C07324=1151.022,358.801,-80.777,-176.348,9.228,148.809
C07325=1151.025,358.554,-80.742,-176.350,9.224,148.808
C07326=1151.029,358.306,-80.708,-176.353,9.220,148.808
C07327=1151.034,358.059,-80.672,-176.355,9.216,148.807
C07328=1151.038,357.811,-80.638,-176.358,9.212,148.807
C07329=1151.041,357.564,-80.602,-176.361,9.208,148.807
C07330=1151.045,357.317,-80.568,-176.363,9.205,148.807
C07331=1151.049,357.068,-80.533,-176.365,9.201,148.806
C07332=1151.053,356.822,-80.498,-176.368,9.196,148.806
C07333=1151.057,356.573,-80.463,-176.370,9.193,148.806
C07334=1151.062,356.326,-80.429,-176.373,9.189,148.805
C07335=1151.065,356.079,-80.394,-176.375,9.185,148.805
C07336=1151.069,355.831,-80.359,-176.378,9.181,148.805
C07337=1151.073,355.583,-80.325,-176.380,9.178,148.804
C07338=1151.076,355.336,-80.290,-176.383,9.173,148.804
C07339=1151.081,355.089,-80.255,-176.386,9.169,148.804
C07340=1151.085,354.841,-80.220,-176.388,9.166,148.804
C07341=1151.089,354.593,-80.186,-176.390,9.162,148.803
C07342=1151.093,354.345,-80.152,-176.393,9.158,148.803
C07343=1151.097,354.099,-80.116,-176.396,9.154,148.803
C07344=1151.101,353.850,-80.082,-176.398,9.151,148.802
C07345=1151.105,353.603,-80.048,-176.400,9.147,148.802
C07346=1151.109,353.355,-80.013,-176.403,9.143,148.802
C07347=1151.113,353.108,-79.978,-176.405,9.139,148.801
C07348=1151.116,352.860,-79.944,-176.408,9.135,148.801
C07349=1151.121,352.613,-79.910,-176.410,9.132,148.801
C07350=1151.124,352.365,-79.875,-176.413,9.127,148.800
C07351=1151.128,352.118,-79.840,-176.415,9.124,148.800
C07352=1151.132,351.870,-79.805,-176.418,9.120,148.800
C07353=1151.136,351.623,-79.772,-176.420,9.116,148.799
C07354=1151.140,351.375,-79.737,-176.423,9.112,148.799
C07355=1151.144,351.127,-79.703,-176.425,9.109,148.799
C07356=1151.149,350.880,-79.668,-176.428,9.105,148.799
C07357=1151.153,350.632,-79.634,-176.431,9.100,148.798
C07358=1151.156,350.385,-79.600,-176.433,9.097,148.798
C07359=1151.160,350.137,-79.565,-176.436,9.093,148.798
C07360=1151.164,349.890,-79.531,-176.438,9.089,148.797
C07361=1151.168,349.641,-79.496,-176.441,9.085,148.797
C07362=1151.172,349.394,-79.463,-176.443,9.082,148.797
C07363=1151.177,349.146,-79.429,-176.446,9.078,148.797
C07364=1151.180,348.899,-79.394,-176.448,9.074,148.796
C07365=1151.185,348.651,-79.360,-176.451,9.070,148.796
C07366=1151.188,348.403,-79.326,-176.453,9.067,148.796
C07367=1151.193,348.156,-79.291,-176.456,9.063,148.796
C07368=1151.196,347.909,-79.257,-176.458,9.059,148.795
C07369=1151.201,347.660,-79.223,-176.461,9.055,148.795
C07370=1151.204,347.413,-79.189,-176.463,9.052,148.795
C07371=1151.209,347.166,-79.155,-176.466,9.048,148.794
C07372=1151.212,346.918,-79.121,-176.468,9.044,148.794
C07373=1151.216,346.670,-79.087,-176.471,9.040,148.794
C07374=1151.221,346.423,-79.053,-176.473,9.037,148.794
C07375=1151.224,346.175,-79.019,-176.476,9.033,148.793
C07376=1151.229,345.927,-78.984,-176.478,9.029,148.793
C07377=1151.233,345.680,-78.951,-176.481,9.025,148.793
C07378=1151.236,345.432,-78.917,-176.483,9.022,148.792
C07379=1151.241,345.184,-78.882,-176.486,9.018,148.792
C07380=1151.245,344.937,-78.849,-176.488,9.014,148.792
C07381=1151.248,344.689,-78.815,-176.491,9.010,148.792
C07382=1151.253,344.441,-78.781,-176.493,9.007,148.791
C07383=1151.257,344.194,-78.747,-176.496,9.003,148.791
C07384=1151.261,343.947,-78.714,-176.498,8.999,148.791
C07385=1151.265,343.698,-78.679,-176.501,8.995,148.790
C07386=1151.269,343.451,-78.646,-176.503,8.992,148.790
C07387=1151.273,343.203,-78.612,-176.506,8.988,148.790
C07388=1151.277,342.955,-78.578,-176.508,8.984,148.790
C07389=1151.281,342.707,-78.544,-176.511,8.980,148.789
C07390=1151.285,342.460,-78.511,-176.514,8.977,148.789
C07391=1151.289,342.212,-78.477,-176.516,8.973,148.789
C07392=1151.293,341.964,-78.443,-176.518,8.969,148.789
C07393=1151.297,341.716,-78.409,-176.521,8.965,148.788
C07394=1151.301,341.469,-78.376,-176.524,8.962,148.788
C07395=1151.305,341.222,-78.342,-176.527,8.958,148.788
C07396=1151.310,340.974,-78.308,-176.529,8.955,148.788
C07397=1151.313,340.726,-78.274,-176.531,8.950,148.787
C07398=1151.317,340.478,-78.241,-176.534,8.947,148.787
C07399=1151.321,340.231,-78.207,-176.536,8.944,148.787
C07400=1151.325,339.983,-78.174,-176.539,8.940,148.787
C07401=1151.330,339.703,-78.136,-176.542,8.936,148.786
C07402=1151.335,339.423,-78.098,-176.545,8.931,148.786
C07403=1151.339,339.142,-78.060,-176.548,8.927,148.786
C07404=1151.344,338.863,-78.022,-176.550,8.923,148.785
C07405=1151.347,338.614,-77.989,-176.553,8.919,148.785
C07406=1151.352,338.367,-77.955,-176.555,8.916,148.785
C07407=1151.355,338.120,-77.922,-176.558,8.912,148.785
C07408=1151.360,337.871,-77.888,-176.560,8.908,148.785
C07409=1151.364,337.624,-77.855,-176.563,8.905,148.784
C07410=1151.369,337.376,-77.822,-176.566,8.901,148.784
C07411=1151.372,337.128,-77.787,-176.568,8.898,148.784
C07412=1151.376,336.880,-77.754,-176.571,8.893,148.784
C07413=1151.380,336.633,-77.721,-176.573,8.890,148.783
C07414=1151.384,336.385,-77.688,-176.575,8.887,148.783
C07415=1151.388,336.137,-77.655,-176.578,8.883,148.783
C07416=1151.392,335.890,-77.622,-176.580,8.879,148.783
C07417=1151.397,335.642,-77.588,-176.583,8.875,148.782
C07418=1151.401,335.394,-77.555,-176.586,8.872,148.782
C07419=1151.405,335.147,-77.521,-176.588,8.868,148.782
C07420=1151.408,334.899,-77.488,-176.591,8.865,148.782
C07421=1151.412,334.651,-77.455,-176.593,8.861,148.782
C07422=1151.416,334.403,-77.422,-176.596,8.857,148.781
C07423=1151.421,334.155,-77.388,-176.598,8.854,148.781
C07424=1151.425,333.908,-77.355,-176.601,8.850,148.781
C07425=1151.429,333.660,-77.322,-176.604,8.847,148.781
C07426=1151.433,333.412,-77.289,-176.606,8.842,148.780
C07427=1151.437,333.164,-77.256,-176.609,8.839,148.780
C07428=1151.440,332.917,-77.223,-176.611,8.836,148.780
C07429=1151.445,332.669,-77.190,-176.614,8.831,148.780
C07430=1151.449,332.421,-77.158,-176.616,8.828,148.779
C07431=1151.453,332.173,-77.124,-176.619,8.824,148.779
C07432=1151.457,331.926,-77.091,-176.621,8.821,148.779
C07433=1151.461,331.678,-77.058,-176.623,8.818,148.779
C07434=1151.466,331.430,-77.025,-176.626,8.813,148.778
C07435=1151.470,331.182,-76.992,-176.629,8.810,148.778
C07436=1151.473,330.935,-76.959,-176.632,8.806,148.778
C07437=1151.478,330.687,-76.927,-176.634,8.803,148.778
C07438=1151.482,330.439,-76.894,-176.636,8.800,148.778
C07439=1151.486,330.191,-76.860,-176.639,8.795,148.777
C07440=1151.490,329.943,-76.827,-176.641,8.792,148.777
C07441=1151.494,329.696,-76.794,-176.644,8.788,148.777
C07442=1151.498,329.448,-76.762,-176.647,8.785,148.777
C07443=1151.502,329.200,-76.729,-176.649,8.782,148.777
C07444=1151.506,328.952,-76.696,-176.652,8.777,148.776
C07445=1151.511,328.704,-76.664,-176.654,8.774,148.776
C07446=1151.514,328.456,-76.631,-176.657,8.770,148.776
C07447=1151.518,328.209,-76.598,-176.659,8.767,148.776
C07448=1151.523,327.960,-76.565,-176.662,8.764,148.775
C07449=1151.527,327.713,-76.532,-176.665,8.759,148.775
C07450=1151.530,327.465,-76.500,-176.667,8.757,148.775
C07451=1151.535,327.217,-76.467,-176.670,8.753,148.775
C07452=1151.539,326.969,-76.434,-176.673,8.749,148.775
C07453=1151.543,326.722,-76.402,-176.675,8.746,148.775
C07454=1151.547,326.474,-76.369,-176.678,8.742,148.774
C07455=1151.551,326.226,-76.336,-176.680,8.739,148.774
C07456=1151.556,325.978,-76.304,-176.682,8.735,148.774
C07457=1151.559,325.731,-76.271,-176.685,8.731,148.774
C07458=1151.564,325.482,-76.239,-176.688,8.728,148.774
C07459=1151.567,325.235,-76.206,-176.690,8.725,148.773
C07460=1151.571,324.986,-76.174,-176.693,8.721,148.773
C07461=1151.576,324.739,-76.141,-176.695,8.717,148.773
C07462=1151.580,324.491,-76.109,-176.698,8.714,148.773
C07463=1151.584,324.244,-76.076,-176.700,8.710,148.773
C07464=1151.588,323.996,-76.044,-176.703,8.707,148.772
C07465=1151.592,323.747,-76.012,-176.706,8.704,148.772
C07466=1151.596,323.499,-75.979,-176.708,8.700,148.772
C07467=1151.600,323.251,-75.947,-176.711,8.696,148.772
C07468=1151.604,323.004,-75.914,-176.713,8.693,148.772
C07469=1151.608,322.756,-75.882,-176.716,8.689,148.771
C07470=1151.613,322.508,-75.850,-176.718,8.686,148.771
C07471=1151.616,322.261,-75.817,-176.721,8.682,148.771
C07472=1151.621,322.012,-75.785,-176.723,8.678,148.771
C07473=1151.624,321.764,-75.753,-176.726,8.675,148.771
C07474=1151.629,321.516,-75.720,-176.729,8.671,148.771
C07475=1151.633,321.269,-75.688,-176.731,8.668,148.770
C07476=1151.637,321.021,-75.656,-176.734,8.665,148.770
C07477=1151.641,320.773,-75.624,-176.737,8.661,148.770
C07478=1151.645,320.525,-75.591,-176.739,8.657,148.770
C07479=1151.649,320.278,-75.559,-176.741,8.654,148.770
C07480=1151.654,320.029,-75.527,-176.744,8.651,148.769
C07481=1151.658,319.781,-75.495,-176.747,8.647,148.769
C07482=1151.661,319.533,-75.463,-176.749,8.644,148.769
C07483=1151.665,319.286,-75.430,-176.752,8.640,148.769
C07484=1151.670,319.038,-75.399,-176.755,8.636,148.769
C07485=1151.674,318.790,-75.366,-176.757,8.633,148.769
C07486=1151.678,318.542,-75.334,-176.759,8.630,148.768
C07487=1151.682,318.294,-75.302,-176.762,8.626,148.768
C07488=1151.687,318.046,-75.270,-176.765,8.623,148.768
C07489=1151.690,317.798,-75.238,-176.767,8.619,148.768
C07490=1151.694,317.550,-75.207,-176.770,8.615,148.768
C07491=1151.699,317.302,-75.175,-176.772,8.612,148.768
C07492=1151.703,317.054,-75.143,-176.775,8.609,148.767
C07493=1151.707,316.806,-75.111,-176.778,8.605,148.767
C07494=1151.712,316.559,-75.079,-176.780,8.602,148.767
C07495=1151.715,316.311,-75.047,-176.783,8.599,148.767
C07496=1151.719,316.063,-75.015,-176.785,8.595,148.767
C07497=1151.723,315.814,-74.983,-176.788,8.591,148.767
C07498=1151.728,315.567,-74.951,-176.791,8.588,148.767
C07499=1151.731,315.319,-74.919,-176.793,8.585,148.766
C07500=1151.736,315.071,-74.887,-176.796,8.581,148.766
C07501=1151.740,314.823,-74.855,-176.798,8.578,148.766
C07502=1151.744,314.575,-74.824,-176.801,8.575,148.766
C07503=1151.748,314.328,-74.792,-176.804,8.571,148.766
C07504=1151.753,314.079,-74.760,-176.806,8.567,148.766
C07505=1151.757,313.802,-74.724,-176.809,8.563,148.765
C07506=1151.762,313.524,-74.689,-176.812,8.560,148.765
C07507=1151.767,313.247,-74.654,-176.815,8.556,148.765
C07508=1151.771,312.969,-74.618,-176.818,8.552,148.765
C07509=1151.775,312.721,-74.586,-176.820,8.549,148.765
C07510=1151.780,312.474,-74.554,-176.823,8.545,148.765
C07511=1151.784,312.225,-74.523,-176.826,8.542,148.765
C07512=1151.788,311.978,-74.492,-176.828,8.538,148.764
C07513=1151.792,311.730,-74.460,-176.830,8.535,148.764
C07514=1151.796,311.481,-74.429,-176.834,8.531,148.764
C07515=1151.800,311.234,-74.397,-176.836,8.528,148.764
C07516=1151.804,310.986,-74.365,-176.838,8.525,148.764
C07517=1151.809,310.738,-74.333,-176.841,8.522,148.764
C07518=1151.813,310.489,-74.302,-176.844,8.518,148.764
C07519=1151.817,310.242,-74.271,-176.846,8.515,148.763
C07520=1151.821,309.993,-74.240,-176.849,8.511,148.763
C07521=1151.825,309.745,-74.208,-176.852,8.507,148.763
C07522=1151.829,309.498,-74.176,-176.854,8.504,148.763
C07523=1151.833,309.249,-74.145,-176.856,8.501,148.763
C07524=1151.837,309.002,-74.114,-176.859,8.498,148.763
C07525=1151.841,308.753,-74.083,-176.862,8.494,148.763
C07526=1151.846,308.506,-74.051,-176.864,8.491,148.762
C07527=1151.850,308.257,-74.020,-176.867,8.488,148.763
C07528=1151.854,308.010,-73.989,-176.870,8.484,148.762
C07529=1151.858,307.761,-73.957,-176.872,8.480,148.762
C07530=1151.862,307.514,-73.926,-176.875,8.477,148.762
C07531=1151.866,307.265,-73.895,-176.878,8.474,148.762
C07532=1151.871,307.018,-73.863,-176.880,8.471,148.762
C07533=1151.875,306.769,-73.832,-176.883,8.467,148.762
C07534=1151.879,306.522,-73.801,-176.886,8.464,148.762
C07535=1151.884,306.274,-73.770,-176.888,8.460,148.761
C07536=1151.887,306.026,-73.738,-176.891,8.458,148.761
C07537=1151.892,305.778,-73.707,-176.893,8.454,148.761
C07538=1151.896,305.529,-73.676,-176.896,8.450,148.761
C07539=1151.900,305.282,-73.645,-176.899,8.447,148.761
C07540=1151.904,305.033,-73.614,-176.901,8.444,148.761
C07541=1151.909,304.785,-73.583,-176.903,8.441,148.761
C07542=1151.913,304.537,-73.551,-176.907,8.437,148.761
C07543=1151.917,304.289,-73.520,-176.909,8.434,148.760
C07544=1151.922,304.041,-73.489,-176.911,8.430,148.760
C07545=1151.925,303.794,-73.458,-176.914,8.427,148.760
C07546=1151.929,303.546,-73.427,-176.917,8.423,148.760
C07547=1151.933,303.297,-73.396,-176.920,8.420,148.760
C07548=1151.938,303.049,-73.366,-176.922,8.417,148.760
C07549=1151.942,302.802,-73.334,-176.924,8.414,148.760
C07550=1151.946,302.553,-73.303,-176.927,8.411,148.760
C07551=1151.951,302.305,-73.272,-176.930,8.407,148.760
C07552=1151.955,302.058,-73.242,-176.933,8.404,148.760
C07553=1151.959,301.809,-73.211,-176.935,8.401,148.759
C07554=1151.963,301.561,-73.180,-176.937,8.397,148.759
C07555=1151.968,301.314,-73.149,-176.940,8.394,148.759
C07556=1151.972,301.065,-73.118,-176.943,8.390,148.759
C07557=1151.976,300.817,-73.087,-176.946,8.387,148.759
C07558=1151.980,300.569,-73.056,-176.948,8.384,148.759
C07559=1151.984,300.321,-73.025,-176.950,8.381,148.759
C07560=1151.989,300.073,-72.995,-176.953,8.378,148.759
C07561=1151.993,299.825,-72.965,-176.956,8.374,148.759
C07562=1151.997,299.576,-72.933,-176.959,8.371,148.759
C07563=1152.001,299.328,-72.903,-176.961,8.367,148.758
C07564=1152.005,299.081,-72.872,-176.964,8.365,148.758
C07565=1152.009,298.832,-72.841,-176.966,8.361,148.758
C07566=1152.014,298.584,-72.811,-176.970,8.357,148.758
C07567=1152.018,298.337,-72.780,-176.972,8.354,148.758
C07568=1152.022,298.088,-72.749,-176.974,8.351,148.758
C07569=1152.026,297.840,-72.718,-176.977,8.348,148.758
C07570=1152.030,297.592,-72.688,-176.979,8.345,148.758
C07571=1152.035,297.344,-72.658,-176.983,8.341,148.758
C07572=1152.039,297.096,-72.626,-176.985,8.338,148.758
C07573=1152.043,296.848,-72.596,-176.988,8.335,148.758
C07574=1152.047,296.600,-72.565,-176.990,8.331,148.757
C07575=1152.052,296.351,-72.535,-176.993,8.328,148.757
C07576=1152.056,296.103,-72.505,-176.995,8.325,148.757
C07577=1152.060,295.855,-72.474,-176.998,8.321,148.757
C07578=1152.064,295.608,-72.444,-177.001,8.318,148.757
C07579=1152.069,295.360,-72.413,-177.004,8.315,148.757
C07580=1152.072,295.111,-72.383,-177.006,8.312,148.757
C07581=1152.077,294.863,-72.353,-177.009,8.309,148.757
C07582=1152.081,294.615,-72.322,-177.012,8.305,148.757
C07583=1152.085,294.367,-72.292,-177.014,8.302,148.757
C07584=1152.089,294.118,-72.261,-177.017,8.299,148.757
C07585=1152.094,293.870,-72.231,-177.019,8.296,148.757
C07586=1152.098,293.622,-72.200,-177.022,8.292,148.757
C07587=1152.102,293.375,-72.170,-177.024,8.290,148.757
C07588=1152.106,293.126,-72.141,-177.027,8.286,148.756
C07589=1152.111,292.878,-72.110,-177.030,8.282,148.756
C07590=1152.114,292.630,-72.079,-177.032,8.279,148.756
C07591=1152.119,292.381,-72.049,-177.035,8.276,148.756
C07592=1152.123,292.134,-72.019,-177.038,8.273,148.756
C07593=1152.127,291.886,-71.988,-177.040,8.270,148.756
C07594=1152.132,291.637,-71.959,-177.043,8.267,148.756
C07595=1152.136,291.390,-71.928,-177.046,8.263,148.756
C07596=1152.140,291.141,-71.898,-177.049,8.260,148.756
C07597=1152.144,290.893,-71.868,-177.051,8.257,148.756
C07598=1152.149,290.644,-71.838,-177.054,8.254,148.756
C07599=1152.153,290.397,-71.808,-177.056,8.251,148.756
C07600=1152.157,290.148,-71.778,-177.059,8.248,148.756
C07601=1152.161,289.900,-71.748,-177.061,8.244,148.756
C07602=1152.165,289.652,-71.718,-177.065,8.241,148.756
C07603=1152.170,289.404,-71.688,-177.067,8.238,148.756
C07604=1152.174,289.156,-71.658,-177.070,8.234,148.755
C07605=1152.178,288.908,-71.628,-177.072,8.231,148.755
C07606=1152.182,288.659,-71.598,-177.075,8.228,148.755
C07607=1152.186,288.411,-71.567,-177.077,8.225,148.755
C07608=1152.191,288.163,-71.538,-177.080,8.222,148.755
C07609=1152.195,287.888,-71.505,-177.083,8.218,148.755
C07610=1152.201,287.613,-71.471,-177.086,8.215,148.755
C07611=1152.205,287.337,-71.438,-177.089,8.211,148.755
C07612=1152.210,287.062,-71.405,-177.092,8.207,148.755
C07613=1152.214,286.814,-71.375,-177.095,8.204,148.755
C07614=1152.218,286.566,-71.346,-177.097,8.201,148.755
C07615=1152.223,286.317,-71.315,-177.100,8.198,148.755
C07616=1152.227,286.070,-71.285,-177.103,8.195,148.755
C07617=1152.231,285.821,-71.256,-177.105,8.192,148.755
C07618=1152.235,285.573,-71.226,-177.108,8.189,148.755
C07619=1152.239,285.325,-71.197,-177.110,8.186,148.755
C07620=1152.244,285.077,-71.166,-177.114,8.182,148.755
C07621=1152.248,284.829,-71.137,-177.116,8.179,148.755
C07622=1152.252,284.580,-71.107,-177.119,8.176,148.755
C07623=1152.256,284.332,-71.078,-177.121,8.173,148.755
C07624=1152.261,284.084,-71.048,-177.124,8.170,148.755
C07625=1152.266,283.835,-71.018,-177.126,8.167,148.754
C07626=1152.269,283.588,-70.988,-177.129,8.164,148.754
C07627=1152.274,283.339,-70.959,-177.132,8.161,148.755
C07628=1152.278,283.091,-70.929,-177.134,8.157,148.754
C07629=1152.282,282.843,-70.900,-177.137,8.154,148.754
C07630=1152.286,282.595,-70.870,-177.140,8.151,148.754
C07631=1152.290,282.346,-70.841,-177.143,8.147,148.754
C07632=1152.294,282.098,-70.811,-177.146,8.145,148.754
C07633=1152.300,281.850,-70.782,-177.148,8.142,148.754
C07634=1152.304,281.602,-70.752,-177.151,8.138,148.754
C07635=1152.308,281.354,-70.723,-177.153,8.135,148.754
C07636=1152.313,281.105,-70.693,-177.156,8.132,148.754
C07637=1152.317,280.857,-70.664,-177.158,8.129,148.754
C07638=1152.321,280.609,-70.634,-177.161,8.126,148.754
C07639=1152.325,280.361,-70.605,-177.164,8.123,148.754
C07640=1152.329,280.112,-70.576,-177.166,8.120,148.754
C07641=1152.333,279.864,-70.546,-177.170,8.116,148.754
C07642=1152.338,279.616,-70.517,-177.172,8.113,148.754
C07643=1152.342,279.367,-70.487,-177.175,8.110,148.754
C07644=1152.347,279.120,-70.458,-177.178,8.107,148.754
C07645=1152.351,278.872,-70.429,-177.180,8.104,148.754
C07646=1152.355,278.623,-70.399,-177.183,8.101,148.754
C07647=1152.359,278.375,-70.370,-177.185,8.098,148.754
C07648=1152.364,278.126,-70.341,-177.188,8.095,148.754
C07649=1152.368,277.878,-70.312,-177.191,8.092,148.754
C07650=1152.372,277.630,-70.282,-177.193,8.089,148.754
C07651=1152.377,277.382,-70.253,-177.196,8.086,148.754
C07652=1152.380,277.134,-70.224,-177.199,8.083,148.754
C07653=1152.385,276.885,-70.195,-177.202,8.080,148.754
C07654=1152.389,276.637,-70.166,-177.204,8.077,148.754
C07655=1152.393,276.389,-70.137,-177.207,8.074,148.754
C07656=1152.397,276.140,-70.107,-177.210,8.070,148.754
C07657=1152.402,275.892,-70.079,-177.213,8.067,148.754
C07658=1152.407,275.644,-70.049,-177.215,8.064,148.754
C07659=1152.411,275.396,-70.020,-177.218,8.061,148.754
C07660=1152.414,275.148,-69.991,-177.221,8.058,148.754
C07661=1152.419,274.899,-69.962,-177.223,8.055,148.754
C07662=1152.423,274.651,-69.933,-177.226,8.052,148.754
C07663=1152.428,274.402,-69.904,-177.229,8.049,148.754
C07664=1152.432,274.154,-69.875,-177.231,8.046,148.754
C07665=1152.436,273.906,-69.845,-177.234,8.043,148.754
C07666=1152.441,273.658,-69.818,-177.236,8.039,148.754
C07667=1152.445,273.410,-69.788,-177.239,8.037,148.754
C07668=1152.449,273.161,-69.759,-177.242,8.034,148.754
C07669=1152.453,272.913,-69.730,-177.245,8.031,148.754
C07670=1152.457,272.665,-69.702,-177.247,8.027,148.754
C07671=1152.462,272.416,-69.673,-177.250,8.024,148.754
C07672=1152.466,272.168,-69.643,-177.253,8.022,148.754
C07673=1152.471,271.919,-69.615,-177.255,8.019,148.754
C07674=1152.475,271.672,-69.586,-177.258,8.016,148.754
C07675=1152.479,271.423,-69.557,-177.260,8.012,148.754
C07676=1152.483,271.175,-69.528,-177.263,8.009,148.754
C07677=1152.488,270.927,-69.500,-177.266,8.006,148.754
C07678=1152.492,270.678,-69.471,-177.269,8.004,148.754
C07679=1152.496,270.430,-69.442,-177.272,8.001,148.754
C07680=1152.501,270.182,-69.414,-177.274,7.997,148.754
C07681=1152.505,269.934,-69.385,-177.277,7.994,148.754
C07682=1152.509,269.685,-69.356,-177.279,7.991,148.754
C07683=1152.514,269.437,-69.328,-177.282,7.988,148.754
C07684=1152.518,269.189,-69.299,-177.285,7.986,148.754
C07685=1152.522,268.940,-69.270,-177.288,7.983,148.754
C07686=1152.527,268.692,-69.242,-177.290,7.979,148.754
C07687=1152.531,268.444,-69.213,-177.293,7.976,148.754
C07688=1152.535,268.195,-69.184,-177.296,7.973,148.754
C07689=1152.540,267.947,-69.156,-177.299,7.970,148.754
C07690=1152.544,267.699,-69.127,-177.302,7.967,148.754
C07691=1152.548,267.450,-69.099,-177.304,7.964,148.754
C07692=1152.553,267.202,-69.070,-177.307,7.961,148.754
C07693=1152.557,266.953,-69.042,-177.310,7.958,148.754
C07694=1152.561,266.706,-69.013,-177.312,7.955,148.754
C07695=1152.566,266.457,-68.984,-177.315,7.952,148.754
C07696=1152.570,266.208,-68.956,-177.318,7.949,148.754
C07697=1152.575,265.960,-68.928,-177.320,7.947,148.754
C07698=1152.578,265.711,-68.900,-177.323,7.944,148.754
C07699=1152.584,265.463,-68.871,-177.325,7.940,148.754
C07700=1152.587,265.215,-68.842,-177.328,7.938,148.754
C07701=1152.592,264.967,-68.814,-177.331,7.935,148.754
C07702=1152.596,264.719,-68.786,-177.333,7.932,148.754
C07703=1152.600,264.470,-68.757,-177.336,7.929,148.754
C07704=1152.605,264.222,-68.729,-177.339,7.926,148.755
C07705=1152.609,263.973,-68.701,-177.342,7.923,148.755
C07706=1152.613,263.725,-68.673,-177.345,7.920,148.755
C07707=1152.618,263.476,-68.644,-177.347,7.917,148.755
C07708=1152.622,263.228,-68.616,-177.350,7.914,148.755
C07709=1152.626,262.980,-68.588,-177.352,7.911,148.755
C07710=1152.631,262.732,-68.560,-177.355,7.908,148.755
C07711=1152.635,262.483,-68.532,-177.358,7.905,148.755
C07712=1152.640,262.235,-68.503,-177.361,7.902,148.755
C07713=1152.645,261.961,-68.473,-177.364,7.898,148.755
C07714=1152.649,261.689,-68.441,-177.367,7.895,148.755
C07715=1152.654,261.415,-68.411,-177.370,7.892,148.755
C07716=1152.659,261.142,-68.379,-177.373,7.888,148.755
C07717=1152.663,260.893,-68.351,-177.376,7.886,148.755
C07718=1152.667,260.645,-68.323,-177.379,7.883,148.755
C07719=1152.672,260.396,-68.295,-177.381,7.880,148.755
C07720=1152.676,260.148,-68.268,-177.384,7.877,148.755
C07721=1152.680,259.899,-68.239,-177.386,7.875,148.755
C07722=1152.685,259.651,-68.211,-177.389,7.872,148.755
C07723=1152.689,259.403,-68.183,-177.392,7.869,148.755
C07724=1152.693,259.155,-68.155,-177.394,7.865,148.755
C07725=1152.698,258.906,-68.126,-177.397,7.863,148.755
C07726=1152.702,258.657,-68.099,-177.400,7.860,148.755
C07727=1152.707,258.409,-68.072,-177.403,7.857,148.755
C07728=1152.711,258.161,-68.043,-177.405,7.854,148.756
C07729=1152.716,257.913,-68.015,-177.408,7.851,148.756
C07730=1152.720,257.663,-67.988,-177.411,7.848,148.756
C07731=1152.724,257.416,-67.960,-177.414,7.845,148.756
C07732=1152.728,257.167,-67.932,-177.416,7.842,148.756
C07733=1152.732,256.919,-67.905,-177.419,7.839,148.756
C07734=1152.737,256.670,-67.876,-177.422,7.836,148.756
C07735=1152.741,256.422,-67.848,-177.425,7.833,148.756
C07736=1152.746,256.173,-67.821,-177.427,7.830,148.756
C07737=1152.750,255.925,-67.793,-177.430,7.827,148.756
C07738=1152.754,255.677,-67.765,-177.432,7.825,148.756
C07739=1152.759,255.428,-67.738,-177.435,7.822,148.756
C07740=1152.763,255.179,-67.709,-177.438,7.819,148.756
C07741=1152.768,254.931,-67.682,-177.441,7.816,148.756
C07742=1152.772,254.683,-67.655,-177.444,7.813,148.756
C07743=1152.776,254.434,-67.626,-177.446,7.810,148.757
C07744=1152.781,254.186,-67.599,-177.449,7.808,148.757
C07745=1152.785,253.938,-67.572,-177.452,7.805,148.757
C07746=1152.789,253.689,-67.544,-177.455,7.802,148.757
C07747=1152.793,253.441,-67.516,-177.457,7.799,148.757
C07748=1152.798,253.193,-67.489,-177.460,7.796,148.757
C07749=1152.802,252.944,-67.461,-177.463,7.793,148.757
C07750=1152.807,252.695,-67.434,-177.465,7.791,148.757
C07751=1152.811,252.447,-67.406,-177.468,7.788,148.757
C07752=1152.816,252.199,-67.379,-177.471,7.785,148.757
C07753=1152.820,251.950,-67.351,-177.474,7.782,148.757
C07754=1152.825,251.702,-67.323,-177.476,7.779,148.757
C07755=1152.829,251.453,-67.296,-177.479,7.776,148.757
C07756=1152.833,251.205,-67.268,-177.482,7.773,148.757
C07757=1152.838,250.956,-67.241,-177.485,7.770,148.757
C07758=1152.842,250.708,-67.214,-177.487,7.767,148.758
C07759=1152.847,250.460,-67.186,-177.490,7.764,148.758
C07760=1152.851,250.211,-67.159,-177.493,7.761,148.758
C07761=1152.855,249.962,-67.132,-177.495,7.759,148.758
C07762=1152.860,249.714,-67.104,-177.498,7.756,148.758
C07763=1152.864,249.466,-67.077,-177.501,7.753,148.758
C07764=1152.868,249.217,-67.050,-177.504,7.750,148.758
C07765=1152.872,248.968,-67.023,-177.506,7.748,148.758
C07766=1152.877,248.720,-66.995,-177.509,7.745,148.758
C07767=1152.881,248.472,-66.968,-177.512,7.742,148.758
C07768=1152.886,248.223,-66.941,-177.515,7.739,148.758
C07769=1152.890,247.974,-66.914,-177.517,7.737,148.759
C07770=1152.895,247.726,-66.887,-177.520,7.734,148.759
C07771=1152.899,247.478,-66.859,-177.523,7.731,148.759
C07772=1152.904,247.229,-66.832,-177.526,7.728,148.759
C07773=1152.908,246.981,-66.805,-177.528,7.725,148.759
C07774=1152.912,246.732,-66.778,-177.531,7.722,148.759
C07775=1152.916,246.484,-66.751,-177.534,7.719,148.759
C07776=1152.921,246.235,-66.724,-177.537,7.716,148.759
C07777=1152.926,245.987,-66.697,-177.539,7.714,148.759
C07778=1152.930,245.739,-66.669,-177.542,7.711,148.759
C07779=1152.935,245.490,-66.642,-177.544,7.708,148.759
C07780=1152.939,245.242,-66.616,-177.547,7.705,148.759
C07781=1152.943,244.993,-66.588,-177.550,7.703,148.759
C07782=1152.947,244.744,-66.561,-177.553,7.700,148.760
C07783=1152.952,244.496,-66.534,-177.556,7.697,148.760
C07784=1152.956,244.248,-66.508,-177.558,7.695,148.760
C07785=1152.960,243.999,-66.480,-177.561,7.692,148.760
C07786=1152.965,243.751,-66.453,-177.564,7.689,148.760
C07787=1152.970,243.502,-66.426,-177.567,7.686,148.760
C07788=1152.974,243.254,-66.400,-177.569,7.683,148.760
C07789=1152.978,243.005,-66.372,-177.572,7.680,148.760
C07790=1152.982,242.756,-66.345,-177.575,7.677,148.760
C07791=1152.987,242.508,-66.318,-177.578,7.675,148.761
C07792=1152.991,242.259,-66.293,-177.580,7.673,148.761
C07793=1152.996,242.010,-66.266,-177.583,7.670,148.761
C07794=1153.001,241.762,-66.238,-177.586,7.667,148.761
C07795=1153.005,241.514,-66.212,-177.589,7.664,148.761
C07796=1153.009,241.265,-66.185,-177.592,7.661,148.761
C07797=1153.014,241.017,-66.158,-177.594,7.659,148.761
C07798=1153.018,240.769,-66.131,-177.597,7.656,148.761
C07799=1153.023,240.519,-66.105,-177.600,7.653,148.762
C07800=1153.027,240.271,-66.078,-177.603,7.650,148.762
C07801=1153.031,240.023,-66.052,-177.605,7.647,148.762
C07802=1153.036,239.774,-66.024,-177.608,7.644,148.762
C07803=1153.040,239.526,-65.998,-177.610,7.642,148.762
C07804=1153.045,239.277,-65.972,-177.613,7.639,148.762
C07805=1153.050,239.029,-65.945,-177.616,7.636,148.762
C07806=1153.053,238.780,-65.918,-177.619,7.634,148.762
C07807=1153.058,238.531,-65.892,-177.622,7.631,148.762
C07808=1153.062,238.283,-65.865,-177.624,7.629,148.763
C07809=1153.067,238.035,-65.838,-177.627,7.626,148.763
C07810=1153.071,237.786,-65.812,-177.630,7.623,148.763
C07811=1153.076,237.537,-65.785,-177.632,7.620,148.763
C07812=1153.080,237.289,-65.759,-177.636,7.617,148.763
C07813=1153.085,237.040,-65.733,-177.638,7.615,148.763
C07814=1153.089,236.792,-65.706,-177.641,7.612,148.763
C07815=1153.093,236.543,-65.679,-177.643,7.609,148.763
C07816=1153.098,236.294,-65.653,-177.646,7.606,148.763
C07817=1153.103,236.023,-65.624,-177.649,7.604,148.764
C07818=1153.108,235.751,-65.595,-177.652,7.601,148.764
C07819=1153.112,235.479,-65.567,-177.655,7.598,148.764
C07820=1153.117,235.207,-65.537,-177.658,7.595,148.764
C07821=1153.121,234.958,-65.511,-177.661,7.592,148.764
C07822=1153.126,234.710,-65.484,-177.664,7.590,148.764
C07823=1153.131,234.462,-65.459,-177.667,7.587,148.764
C07824=1153.135,234.213,-65.432,-177.669,7.584,148.764
C07825=1153.140,233.964,-65.406,-177.672,7.582,148.765
C07826=1153.144,233.716,-65.379,-177.675,7.579,148.765
C07827=1153.148,233.467,-65.353,-177.678,7.576,148.765
C07828=1153.153,233.218,-65.327,-177.680,7.573,148.765
C07829=1153.157,232.970,-65.301,-177.683,7.571,148.765
C07830=1153.162,232.721,-65.274,-177.685,7.568,148.765
C07831=1153.166,232.473,-65.248,-177.689,7.565,148.766
C07832=1153.170,232.225,-65.223,-177.691,7.563,148.766
C07833=1153.175,231.976,-65.196,-177.694,7.560,148.766
C07834=1153.179,231.727,-65.170,-177.696,7.558,148.766
C07835=1153.183,231.479,-65.144,-177.700,7.555,148.766
C07836=1153.188,231.229,-65.118,-177.702,7.552,148.766
C07837=1153.192,230.981,-65.091,-177.705,7.549,148.766
C07838=1153.197,230.733,-65.066,-177.707,7.547,148.766
C07839=1153.202,230.484,-65.040,-177.710,7.544,148.766
C07840=1153.206,230.236,-65.013,-177.713,7.541,148.767
C07841=1153.210,229.987,-64.987,-177.716,7.539,148.767
C07842=1153.215,229.738,-64.961,-177.718,7.536,148.767
C07843=1153.219,229.489,-64.935,-177.721,7.533,148.767
C07844=1153.224,229.242,-64.909,-177.724,7.531,148.767
C07845=1153.228,228.993,-64.883,-177.727,7.528,148.767
C07846=1153.233,228.744,-64.857,-177.729,7.526,148.768
C07847=1153.237,228.495,-64.831,-177.732,7.523,148.768
C07848=1153.242,228.247,-64.806,-177.735,7.520,148.768
C07849=1153.246,227.998,-64.780,-177.738,7.517,148.768
C07850=1153.250,227.750,-64.754,-177.740,7.515,148.768
C07851=1153.255,227.501,-64.727,-177.743,7.512,148.768
C07852=1153.260,227.252,-64.702,-177.747,7.510,148.769
C07853=1153.264,227.004,-64.676,-177.749,7.508,148.769
C07854=1153.269,226.755,-64.650,-177.752,7.505,148.769
C07855=1153.273,226.506,-64.625,-177.754,7.502,148.769
C07856=1153.277,226.257,-64.599,-177.758,7.499,148.769
C07857=1153.282,226.009,-64.574,-177.760,7.497,148.769
C07858=1153.287,225.760,-64.547,-177.763,7.494,148.769
C07859=1153.291,225.511,-64.521,-177.766,7.492,148.770
C07860=1153.296,225.263,-64.496,-177.769,7.489,148.770
C07861=1153.300,225.014,-64.470,-177.771,7.487,148.770
C07862=1153.304,224.766,-64.445,-177.774,7.484,148.770
C07863=1153.309,224.517,-64.419,-177.777,7.481,148.770
C07864=1153.313,224.269,-64.393,-177.779,7.479,148.770
C07865=1153.318,224.020,-64.368,-177.782,7.476,148.770
C07866=1153.322,223.771,-64.342,-177.785,7.473,148.771
C07867=1153.327,223.523,-64.317,-177.787,7.471,148.771
C07868=1153.331,223.274,-64.291,-177.790,7.468,148.771
C07869=1153.335,223.025,-64.265,-177.793,7.466,148.771
C07870=1153.341,222.777,-64.239,-177.796,7.463,148.771
C07871=1153.345,222.528,-64.213,-177.798,7.461,148.771
C07872=1153.349,222.279,-64.188,-177.801,7.458,148.772
C07873=1153.354,222.031,-64.163,-177.804,7.455,148.772
C07874=1153.358,221.782,-64.137,-177.807,7.453,148.772
C07875=1153.363,221.533,-64.111,-177.809,7.450,148.772
C07876=1153.368,221.285,-64.086,-177.813,7.448,148.772
C07877=1153.371,221.036,-64.062,-177.815,7.445,148.772
C07878=1153.376,220.788,-64.036,-177.818,7.443,148.773
C07879=1153.380,220.539,-64.010,-177.821,7.440,148.773
C07880=1153.385,220.290,-63.985,-177.823,7.438,148.773
C07881=1153.389,220.042,-63.959,-177.826,7.435,148.773
C07882=1153.394,219.793,-63.934,-177.829,7.432,148.773
C07883=1153.399,219.545,-63.909,-177.831,7.430,148.774
C07884=1153.403,219.296,-63.883,-177.834,7.427,148.774
C07885=1153.408,219.046,-63.858,-177.837,7.425,148.774
C07886=1153.412,218.798,-63.833,-177.840,7.423,148.774
C07887=1153.417,218.549,-63.807,-177.842,7.420,148.774
C07888=1153.422,218.301,-63.782,-177.846,7.417,148.774
C07889=1153.425,218.052,-63.757,-177.848,7.415,148.775
C07890=1153.429,217.803,-63.731,-177.851,7.412,148.775
C07891=1153.435,217.555,-63.707,-177.854,7.410,148.775
C07892=1153.439,217.306,-63.681,-177.856,7.407,148.775
C07893=1153.444,217.057,-63.656,-177.859,7.404,148.775
C07894=1153.448,216.808,-63.631,-177.862,7.402,148.775
C07895=1153.452,216.561,-63.606,-177.864,7.400,148.776
C07896=1153.457,216.311,-63.581,-177.868,7.397,148.776
C07897=1153.462,216.063,-63.555,-177.870,7.394,148.776
C07898=1153.466,215.814,-63.530,-177.873,7.392,148.776
C07899=1153.471,215.565,-63.505,-177.876,7.390,148.776
C07900=1153.475,215.316,-63.480,-177.878,7.387,148.777
C07901=1153.480,215.068,-63.455,-177.881,7.385,148.777
C07902=1153.484,214.819,-63.430,-177.884,7.382,148.777
C07903=1153.489,214.571,-63.405,-177.886,7.380,148.777
C07904=1153.493,214.322,-63.380,-177.889,7.377,148.777
C07905=1153.498,214.073,-63.355,-177.892,7.374,148.778
C07906=1153.502,213.824,-63.330,-177.894,7.372,148.778
C07907=1153.506,213.576,-63.306,-177.898,7.370,148.778
C07908=1153.511,213.327,-63.280,-177.900,7.368,148.778
C07909=1153.516,213.078,-63.255,-177.903,7.365,148.778
C07910=1153.520,212.829,-63.230,-177.906,7.362,148.778
C07911=1153.524,212.581,-63.205,-177.908,7.360,148.779
C07912=1153.529,212.331,-63.180,-177.911,7.357,148.779
C07913=1153.534,212.083,-63.155,-177.914,7.354,148.779
C07914=1153.538,211.835,-63.131,-177.917,7.353,148.779
C07915=1153.543,211.586,-63.106,-177.920,7.350,148.779
C07916=1153.548,211.337,-63.081,-177.922,7.348,148.780
C07917=1153.551,211.088,-63.056,-177.925,7.345,148.780
C07918=1153.556,210.840,-63.031,-177.928,7.342,148.780
C07919=1153.560,210.590,-63.007,-177.931,7.340,148.780
C07920=1153.565,210.342,-62.982,-177.933,7.337,148.780
C07921=1153.570,210.072,-62.955,-177.937,7.335,148.781
C07922=1153.575,209.801,-62.928,-177.939,7.332,148.781
C07923=1153.580,209.531,-62.901,-177.942,7.330,148.781
C07924=1153.585,209.260,-62.875,-177.945,7.327,148.781
C07925=1153.590,209.012,-62.849,-177.948,7.325,148.782
C07926=1153.593,208.762,-62.825,-177.951,7.322,148.782
C07927=1153.599,208.514,-62.800,-177.954,7.320,148.782
C07928=1153.604,208.265,-62.776,-177.956,7.317,148.782
C07929=1153.607,208.016,-62.751,-177.959,7.315,148.782
C07930=1153.613,207.767,-62.726,-177.962,7.312,148.783
C07931=1153.617,207.519,-62.702,-177.964,7.310,148.783
C07932=1153.621,207.270,-62.677,-177.967,7.308,148.783
C07933=1153.626,207.022,-62.653,-177.970,7.305,148.783
C07934=1153.631,206.773,-62.628,-177.973,7.303,148.783
C07935=1153.635,206.524,-62.603,-177.976,7.300,148.784
C07936=1153.640,206.275,-62.579,-177.978,7.298,148.784
C07937=1153.644,206.027,-62.555,-177.981,7.295,148.784
C07938=1153.649,205.777,-62.530,-177.984,7.294,148.784
C07939=1153.653,205.529,-62.506,-177.987,7.291,148.784
C07940=1153.657,205.280,-62.482,-177.989,7.289,148.785
C07941=1153.663,205.032,-62.457,-177.992,7.286,148.785
C07942=1153.666,204.782,-62.432,-177.995,7.283,148.785
C07943=1153.671,204.534,-62.408,-177.998,7.281,148.785
C07944=1153.676,204.285,-62.384,-178.000,7.279,148.785
C07945=1153.680,204.036,-62.359,-178.003,7.277,148.786
C07946=1153.685,203.787,-62.335,-178.006,7.274,148.786
C07947=1153.689,203.538,-62.311,-178.008,7.272,148.786
C07948=1153.695,203.290,-62.287,-178.011,7.269,148.786
C07949=1153.698,203.041,-62.262,-178.014,7.267,148.787
C07950=1153.703,202.792,-62.238,-178.017,7.264,148.787
C07951=1153.708,202.543,-62.213,-178.019,7.263,148.787
C07952=1153.712,202.295,-62.189,-178.022,7.260,148.787
C07953=1153.716,202.046,-62.165,-178.025,7.257,148.788
C07954=1153.722,201.797,-62.141,-178.028,7.255,148.788
C07955=1153.726,201.548,-62.117,-178.031,7.253,148.788
C07956=1153.730,201.300,-62.093,-178.033,7.250,148.788
C07957=1153.735,201.051,-62.068,-178.036,7.248,148.789
C07958=1153.739,200.802,-62.044,-178.039,7.246,148.789
C07959=1153.744,200.553,-62.020,-178.042,7.243,148.789
C07960=1153.748,200.305,-61.996,-178.044,7.241,148.789
C07961=1153.753,200.056,-61.972,-178.047,7.239,148.789
C07962=1153.758,199.807,-61.947,-178.050,7.236,148.790
C07963=1153.762,199.558,-61.924,-178.053,7.234,148.790
C07964=1153.766,199.309,-61.900,-178.055,7.232,148.790
C07965=1153.771,199.061,-61.875,-178.058,7.229,148.790
C07966=1153.776,198.811,-61.852,-178.061,7.227,148.791
C07967=1153.781,198.563,-61.828,-178.064,7.224,148.791
C07968=1153.785,198.315,-61.803,-178.066,7.223,148.791
C07969=1153.789,198.065,-61.780,-178.069,7.220,148.791
C07970=1153.794,197.816,-61.755,-178.072,7.218,148.792
C07971=1153.799,197.567,-61.732,-178.075,7.215,148.792
C07972=1153.803,197.319,-61.708,-178.077,7.213,148.792
C07973=1153.808,197.070,-61.684,-178.080,7.210,148.792
C07974=1153.812,196.821,-61.660,-178.083,7.209,148.793
C07975=1153.818,196.573,-61.636,-178.086,7.206,148.793
C07976=1153.822,196.323,-61.612,-178.088,7.204,148.793
C07977=1153.826,196.074,-61.588,-178.092,7.201,148.793
C07978=1153.831,195.825,-61.564,-178.094,7.199,148.793
C07979=1153.835,195.577,-61.540,-178.097,7.197,148.794
C07980=1153.840,195.328,-61.517,-178.099,7.195,148.794
C07981=1153.844,195.080,-61.493,-178.103,7.192,148.794
C07982=1153.849,194.831,-61.470,-178.105,7.190,148.794
C07983=1153.853,194.582,-61.445,-178.108,7.187,148.795
C07984=1153.859,194.333,-61.422,-178.110,7.185,148.795
C07985=1153.863,194.084,-61.397,-178.114,7.183,148.795
C07986=1153.868,193.835,-61.374,-178.116,7.181,148.796
C07987=1153.872,193.587,-61.350,-178.119,7.178,148.796
C07988=1153.877,193.338,-61.327,-178.122,7.176,148.796
C07989=1153.882,193.089,-61.303,-178.124,7.174,148.796
C07990=1153.885,192.840,-61.279,-178.127,7.172,148.796
C07991=1153.890,192.591,-61.255,-178.130,7.170,148.797
C07992=1153.895,192.342,-61.232,-178.133,7.167,148.797
C07993=1153.899,192.093,-61.208,-178.135,7.165,148.797
C07994=1153.904,191.844,-61.185,-178.138,7.162,148.797
C07995=1153.909,191.595,-61.161,-178.141,7.161,148.798
C07996=1153.913,191.347,-61.137,-178.144,7.158,148.798
C07997=1153.918,191.098,-61.114,-178.146,7.156,148.798
C07998=1153.922,190.849,-61.091,-178.150,7.153,148.799
C07999=1153.927,190.600,-61.066,-178.152,7.151,148.799
C08000=1153.931,190.351,-61.043,-178.155,7.150,148.799
C08001=1153.936,190.102,-61.020,-178.157,7.147,148.799
C08002=1153.941,189.853,-60.996,-178.160,7.145,148.800
C08003=1153.946,189.604,-60.973,-178.163,7.142,148.800
C08004=1153.950,189.357,-60.950,-178.165,7.140,148.800
C08005=1153.955,189.108,-60.927,-178.169,7.138,148.800
C08006=1153.959,188.859,-60.903,-178.171,7.136,148.801
C08007=1153.964,188.610,-60.880,-178.174,7.134,148.801
C08008=1153.969,188.361,-60.856,-178.177,7.131,148.801
C08009=1153.973,188.112,-60.833,-178.179,7.129,148.801
C08010=1153.978,187.863,-60.809,-178.182,7.127,148.802
C08011=1153.982,187.614,-60.786,-178.185,7.125,148.802
C08012=1153.987,187.365,-60.762,-178.188,7.122,148.802
C08013=1153.991,187.116,-60.740,-178.191,7.120,148.802
C08014=1153.996,186.867,-60.716,-178.193,7.118,148.803
C08015=1154.001,186.618,-60.693,-178.196,7.115,148.803
C08016=1154.005,186.369,-60.669,-178.199,7.114,148.803
C08017=1154.010,186.120,-60.646,-178.202,7.111,148.804
C08018=1154.014,185.872,-60.624,-178.204,7.109,148.804
C08019=1154.019,185.623,-60.600,-178.207,7.107,148.804
C08020=1154.024,185.374,-60.577,-178.210,7.104,148.804
C08021=1154.029,185.125,-60.554,-178.212,7.103,148.805
C08022=1154.033,184.876,-60.530,-178.216,7.100,148.805
C08023=1154.037,184.627,-60.508,-178.218,7.098,148.805
C08024=1154.042,184.378,-60.484,-178.221,7.095,148.805
C08025=1154.047,184.109,-60.459,-178.224,7.094,148.806
C08026=1154.052,183.839,-60.433,-178.227,7.091,148.806
C08027=1154.057,183.570,-60.409,-178.230,7.089,148.806
C08028=1154.062,183.300,-60.384,-178.233,7.086,148.807
C08029=1154.067,183.051,-60.361,-178.236,7.084,148.807
C08030=1154.071,182.802,-60.338,-178.239,7.082,148.807
C08031=1154.076,182.553,-60.314,-178.241,7.080,148.807
C08032=1154.081,182.305,-60.292,-178.244,7.078,148.808
C08033=1154.085,182.056,-60.269,-178.247,7.076,148.808
C08034=1154.090,181.807,-60.246,-178.250,7.073,148.808
C08035=1154.094,181.558,-60.223,-178.252,7.071,148.809
C08036=1154.098,181.309,-60.200,-178.255,7.069,148.809
C08037=1154.104,181.061,-60.177,-178.258,7.066,148.809
C08038=1154.109,180.811,-60.154,-178.260,7.065,148.809
C08039=1154.113,180.562,-60.132,-178.263,7.063,148.810
C08040=1154.117,180.313,-60.108,-178.266,7.060,148.810
C08041=1154.121,180.065,-60.085,-178.269,7.058,148.810
C08042=1154.127,179.816,-60.063,-178.271,7.057,148.811
C08043=1154.132,179.567,-60.040,-178.275,7.054,148.811
C08044=1154.136,179.318,-60.017,-178.277,7.052,148.811
C08045=1154.141,179.068,-59.994,-178.280,7.049,148.811
C08046=1154.145,178.820,-59.972,-178.283,7.048,148.812
C08047=1154.150,178.571,-59.949,-178.285,7.045,148.812
C08048=1154.154,178.322,-59.926,-178.288,7.043,148.812
C08049=1154.159,178.073,-59.903,-178.291,7.041,148.813
C08050=1154.164,177.824,-59.880,-178.294,7.039,148.813
C08051=1154.168,177.575,-59.858,-178.296,7.037,148.813
C08052=1154.173,177.326,-59.835,-178.299,7.035,148.814
C08053=1154.177,177.077,-59.812,-178.302,7.033,148.814
C08054=1154.183,176.828,-59.790,-178.305,7.030,148.814
C08055=1154.187,176.580,-59.767,-178.307,7.028,148.814
C08056=1154.192,176.330,-59.744,-178.310,7.027,148.815
C08057=1154.196,176.082,-59.722,-178.313,7.024,148.815
C08058=1154.201,175.833,-59.699,-178.316,7.022,148.815
C08059=1154.205,175.584,-59.677,-178.318,7.020,148.816
C08060=1154.210,175.336,-59.654,-178.321,7.018,148.816
C08061=1154.215,175.086,-59.631,-178.324,7.016,148.816
C08062=1154.219,174.837,-59.609,-178.326,7.014,148.816
C08063=1154.224,174.588,-59.586,-178.330,7.011,148.817
C08064=1154.228,174.340,-59.564,-178.332,7.010,148.817
C08065=1154.233,174.090,-59.541,-178.335,7.008,148.818
C08066=1154.238,173.842,-59.519,-178.338,7.005,148.818
C08067=1154.243,173.592,-59.496,-178.341,7.003,148.818
C08068=1154.247,173.343,-59.474,-178.343,7.001,148.818
C08069=1154.252,173.095,-59.452,-178.347,6.999,148.819
C08070=1154.257,172.845,-59.429,-178.349,6.997,148.819
C08071=1154.261,172.596,-59.406,-178.351,6.995,148.819
C08072=1154.266,172.348,-59.384,-178.354,6.993,148.820
C08073=1154.271,172.098,-59.362,-178.357,6.991,148.820
C08074=1154.275,171.850,-59.339,-178.360,6.989,148.820
C08075=1154.279,171.601,-59.317,-178.362,6.987,148.821
C08076=1154.284,171.351,-59.295,-178.366,6.984,148.821
C08077=1154.289,171.103,-59.272,-178.368,6.983,148.821
C08078=1154.293,170.854,-59.250,-178.371,6.981,148.821
C08079=1154.299,170.605,-59.228,-178.374,6.978,148.822
C08080=1154.303,170.356,-59.205,-178.376,6.976,148.822
C08081=1154.307,170.107,-59.183,-178.379,6.974,148.822
C08082=1154.313,169.858,-59.161,-178.382,6.973,148.823
C08083=1154.317,169.609,-59.139,-178.385,6.970,148.823
C08084=1154.322,169.360,-59.116,-178.387,6.968,148.823
C08085=1154.327,169.111,-59.094,-178.390,6.966,148.824
C08086=1154.331,168.862,-59.072,-178.393,6.964,148.824
C08087=1154.336,168.613,-59.050,-178.396,6.962,148.824
C08088=1154.341,168.364,-59.028,-178.398,6.960,148.825
C08089=1154.345,168.115,-59.005,-178.401,6.958,148.825
C08090=1154.350,167.867,-58.983,-178.404,6.956,148.825
C08091=1154.354,167.617,-58.961,-178.407,6.954,148.826
C08092=1154.359,167.368,-58.939,-178.409,6.952,148.826
C08093=1154.364,167.119,-58.918,-178.412,6.950,148.826
C08094=1154.369,166.870,-58.895,-178.415,6.948,148.827
C08095=1154.373,166.621,-58.873,-178.418,6.946,148.827
C08096=1154.377,166.372,-58.851,-178.421,6.944,148.827
C08097=1154.382,166.124,-58.829,-178.423,6.941,148.827
C08098=1154.387,165.875,-58.807,-178.426,6.939,148.828
C08099=1154.391,165.626,-58.785,-178.429,6.938,148.828
C08100=1154.397,165.377,-58.763,-178.431,6.936,148.829
C08101=1154.401,165.127,-58.741,-178.435,6.933,148.829
C08102=1154.406,164.879,-58.719,-178.437,6.932,148.829
C08103=1154.410,164.629,-58.697,-178.440,6.930,148.829
C08104=1154.415,164.381,-58.675,-178.442,6.928,148.830
C08105=1154.419,164.131,-58.653,-178.446,6.925,148.830
C08106=1154.424,163.883,-58.632,-178.448,6.924,148.831
C08107=1154.429,163.633,-58.610,-178.451,6.922,148.831
C08108=1154.434,163.385,-58.588,-178.453,6.920,148.831
C08109=1154.438,163.135,-58.566,-178.456,6.918,148.831
C08110=1154.443,162.887,-58.544,-178.459,6.915,148.832
C08111=1154.448,162.638,-58.522,-178.462,6.914,148.832
C08112=1154.453,162.388,-58.500,-178.465,6.912,148.833
C08113=1154.457,162.140,-58.478,-178.467,6.910,148.833
C08114=1154.462,161.890,-58.457,-178.471,6.908,148.833
C08115=1154.467,161.641,-58.435,-178.473,6.906,148.833
C08116=1154.471,161.392,-58.413,-178.476,6.904,148.834
C08117=1154.476,161.143,-58.391,-178.478,6.902,148.834
C08118=1154.481,160.895,-58.370,-178.481,6.900,148.835
C08119=1154.485,160.645,-58.348,-178.484,6.898,148.835
C08120=1154.490,160.396,-58.327,-178.487,6.896,148.835
C08121=1154.495,160.147,-58.305,-178.489,6.894,148.835
C08122=1154.499,159.898,-58.283,-178.492,6.892,148.836
C08123=1154.504,159.649,-58.261,-178.495,6.890,148.836
C08124=1154.509,159.400,-58.239,-178.498,6.888,148.837
C08125=1154.513,159.151,-58.219,-178.500,6.886,148.837
C08126=1154.518,158.902,-58.197,-178.503,6.885,148.837
C08127=1154.522,158.653,-58.175,-178.506,6.883,148.838
C08128=1154.527,158.404,-58.153,-178.509,6.880,148.838
C08129=1154.532,158.135,-58.130,-178.512,6.879,148.838
C08130=1154.537,157.866,-58.107,-178.515,6.876,148.839
C08131=1154.542,157.597,-58.083,-178.518,6.874,148.839
C08132=1154.547,157.328,-58.061,-178.521,6.873,148.840
C08133=1154.552,157.079,-58.040,-178.524,6.870,148.840
C08134=1154.557,156.830,-58.018,-178.526,6.868,148.840
C08135=1154.561,156.581,-57.996,-178.529,6.866,148.840
C08136=1154.567,156.332,-57.975,-178.531,6.864,148.841
C08137=1154.572,156.083,-57.953,-178.534,6.863,148.841
C08138=1154.576,155.835,-57.932,-178.537,6.860,148.842
C08139=1154.580,155.585,-57.911,-178.540,6.858,148.842
C08140=1154.585,155.336,-57.889,-178.543,6.857,148.842
C08141=1154.590,155.087,-57.868,-178.546,6.855,148.843
C08142=1154.595,154.838,-57.846,-178.548,6.853,148.843
C08143=1154.600,154.588,-57.825,-178.551,6.851,148.843
C08144=1154.604,154.340,-57.804,-178.554,6.849,148.844
C08145=1154.609,154.091,-57.782,-178.556,6.847,148.844
C08146=1154.613,153.841,-57.761,-178.559,6.845,148.844
C08147=1154.618,153.593,-57.739,-178.562,6.843,148.845
C08148=1154.623,153.343,-57.718,-178.565,6.842,148.845
C08149=1154.627,153.095,-57.697,-178.567,6.840,148.845
C08150=1154.633,152.846,-57.676,-178.571,6.837,148.846
C08151=1154.637,152.596,-57.655,-178.573,6.836,148.846
C08152=1154.642,152.347,-57.633,-178.576,6.834,148.847
C08153=1154.647,152.098,-57.613,-178.578,6.832,148.847
C08154=1154.651,151.850,-57.591,-178.581,6.830,148.847
C08155=1154.656,151.600,-57.570,-178.584,6.828,148.847
C08156=1154.660,151.351,-57.549,-178.587,6.826,148.848
C08157=1154.665,151.102,-57.528,-178.590,6.824,148.848
C08158=1154.670,150.853,-57.507,-178.592,6.822,148.849
C08159=1154.675,150.604,-57.485,-178.595,6.821,148.849
C08160=1154.680,150.355,-57.465,-178.598,6.819,148.849
C08161=1154.684,150.105,-57.443,-178.600,6.817,148.850
C08162=1154.689,149.857,-57.422,-178.603,6.816,148.850
C08163=1154.694,149.608,-57.401,-178.606,6.813,148.851
C08164=1154.699,149.358,-57.380,-178.609,6.811,148.851
C08165=1154.703,149.110,-57.359,-178.612,6.810,148.851
C08166=1154.708,148.861,-57.338,-178.615,6.808,148.852
C08167=1154.713,148.611,-57.317,-178.617,6.806,148.852
C08168=1154.717,148.362,-57.297,-178.619,6.804,148.852
C08169=1154.722,148.113,-57.275,-178.622,6.802,148.853
C08170=1154.727,147.864,-57.254,-178.625,6.801,148.853
C08171=1154.732,147.615,-57.234,-178.628,6.798,148.853
C08172=1154.737,147.366,-57.213,-178.631,6.796,148.854
C08173=1154.741,147.118,-57.192,-178.634,6.795,148.854
C08174=1154.746,146.868,-57.171,-178.636,6.793,148.854
C08175=1154.750,146.619,-57.150,-178.639,6.791,148.855
C08176=1154.755,146.369,-57.129,-178.642,6.789,148.855
C08177=1154.760,146.120,-57.109,-178.644,6.788,148.856
C08178=1154.765,145.871,-57.088,-178.647,6.786,148.856
C08179=1154.770,145.623,-57.066,-178.650,6.784,148.856
C08180=1154.774,145.374,-57.046,-178.653,6.782,148.857
C08181=1154.779,145.124,-57.025,-178.656,6.780,148.857
C08182=1154.784,144.875,-57.004,-178.659,6.778,148.858
C08183=1154.789,144.626,-56.983,-178.661,6.776,148.858
C08184=1154.793,144.377,-56.963,-178.664,6.775,148.858
C08185=1154.798,144.128,-56.942,-178.667,6.773,148.859
C08186=1154.803,143.879,-56.922,-178.669,6.771,148.859
C08187=1154.807,143.630,-56.901,-178.672,6.770,148.859
C08188=1154.812,143.381,-56.880,-178.675,6.768,148.860
C08189=1154.816,143.131,-56.859,-178.677,6.766,148.860
C08190=1154.821,142.882,-56.838,-178.680,6.764,148.861
C08191=1154.826,142.633,-56.818,-178.683,6.762,148.861
C08192=1154.831,142.384,-56.797,-178.686,6.760,148.861
C08193=1154.836,142.135,-56.777,-178.689,6.758,148.862
C08194=1154.840,141.886,-56.756,-178.692,6.757,148.862
C08195=1154.845,141.636,-56.735,-178.694,6.755,148.863
C08196=1154.850,141.388,-56.715,-178.697,6.753,148.863
C08197=1154.855,141.138,-56.694,-178.700,6.752,148.863
C08198=1154.859,140.889,-56.674,-178.702,6.750,148.864
C08199=1154.864,140.640,-56.653,-178.705,6.748,148.864
C08200=1154.869,140.391,-56.632,-178.708,6.746,148.865
C08201=1154.873,140.142,-56.612,-178.711,6.745,148.865
C08202=1154.878,139.893,-56.592,-178.713,6.743,148.865
C08203=1154.883,139.644,-56.571,-178.716,6.741,148.866
C08204=1154.888,139.394,-56.551,-178.719,6.740,148.866
C08205=1154.892,139.145,-56.531,-178.721,6.738,148.866
C08206=1154.898,138.897,-56.510,-178.725,6.735,148.867
C08207=1154.902,138.648,-56.490,-178.727,6.734,148.867
C08208=1154.907,138.399,-56.469,-178.730,6.732,148.868
C08209=1154.912,138.149,-56.449,-178.733,6.730,148.868
C08210=1154.917,137.900,-56.429,-178.736,6.728,148.868
C08211=1154.921,137.651,-56.408,-178.738,6.727,148.869
C08212=1154.926,137.402,-56.387,-178.741,6.725,148.869
C08213=1154.931,137.153,-56.367,-178.744,6.723,148.870
C08214=1154.935,136.903,-56.347,-178.746,6.721,148.870
C08215=1154.940,136.654,-56.327,-178.749,6.720,148.870
C08216=1154.945,136.405,-56.306,-178.752,6.718,148.871
C08217=1154.950,136.156,-56.286,-178.754,6.716,148.871
C08218=1154.954,135.907,-56.266,-178.757,6.715,148.872
C08219=1154.959,135.658,-56.246,-178.760,6.713,148.872
C08220=1154.964,135.410,-56.226,-178.763,6.711,148.872
C08221=1154.969,135.160,-56.205,-178.765,6.709,148.873
C08222=1154.974,134.911,-56.185,-178.768,6.708,148.873
C08223=1154.978,134.661,-56.165,-178.771,6.706,148.873
C08224=1154.983,134.412,-56.145,-178.773,6.704,148.874
C08225=1154.987,134.163,-56.125,-178.776,6.703,148.874
C08226=1154.993,133.913,-56.104,-178.779,6.701,148.875
C08227=1154.998,133.665,-56.084,-178.782,6.699,148.875
C08228=1155.002,133.416,-56.064,-178.784,6.697,148.875
C08229=1155.007,133.167,-56.044,-178.787,6.696,148.876
C08230=1155.011,132.918,-56.024,-178.790,6.694,148.876
C08231=1155.016,132.668,-56.004,-178.792,6.692,148.877
C08232=1155.020,132.419,-55.984,-178.796,6.691,148.877
C08233=1155.026,132.150,-55.962,-178.799,6.688,148.878
C08234=1155.032,131.882,-55.941,-178.802,6.687,148.878
C08235=1155.037,131.614,-55.919,-178.804,6.685,148.878
C08236=1155.042,131.345,-55.898,-178.807,6.683,148.879
C08237=1155.046,131.096,-55.878,-178.810,6.682,148.879
C08238=1155.051,130.847,-55.858,-178.813,6.680,148.880
C08239=1155.056,130.598,-55.838,-178.816,6.678,148.880
C08240=1155.061,130.348,-55.817,-178.818,6.677,148.881
C08241=1155.066,130.099,-55.798,-178.821,6.675,148.881
C08242=1155.071,129.850,-55.778,-178.824,6.673,148.881
C08243=1155.076,129.600,-55.758,-178.827,6.672,148.882
C08244=1155.080,129.352,-55.738,-178.829,6.670,148.882
C08245=1155.085,129.103,-55.718,-178.832,6.668,148.883
C08246=1155.090,128.853,-55.699,-178.835,6.666,148.883
C08247=1155.094,128.604,-55.678,-178.837,6.665,148.883
C08248=1155.099,128.355,-55.659,-178.840,6.663,148.884
C08249=1155.104,128.106,-55.639,-178.843,6.661,148.884
C08250=1155.109,127.857,-55.619,-178.846,6.660,148.885
C08251=1155.114,127.607,-55.599,-178.848,6.658,148.885
C08252=1155.118,127.358,-55.579,-178.851,6.657,148.886
C08253=1155.124,127.109,-55.560,-178.854,6.655,148.886
C08254=1155.128,126.860,-55.540,-178.857,6.653,148.886
C08255=1155.133,126.610,-55.520,-178.860,6.651,148.887
C08256=1155.137,126.361,-55.500,-178.862,6.650,148.887
C08257=1155.142,126.113,-55.481,-178.865,6.648,148.888
C08258=1155.147,125.863,-55.462,-178.868,6.646,148.888
C08259=1155.152,125.614,-55.442,-178.870,6.645,148.888
C08260=1155.157,125.365,-55.422,-178.873,6.643,148.889
C08261=1155.161,125.116,-55.402,-178.876,6.641,148.889
C08262=1155.166,124.866,-55.383,-178.879,6.640,148.890
C08263=1155.171,124.617,-55.363,-178.882,6.638,148.890
C08264=1155.176,124.368,-55.343,-178.884,6.637,148.891
C08265=1155.181,124.119,-55.323,-178.887,6.635,148.891
C08266=1155.185,123.870,-55.305,-178.889,6.634,148.891
C08267=1155.190,123.621,-55.285,-178.892,6.632,148.892
C08268=1155.195,123.371,-55.265,-178.895,6.630,148.892
C08269=1155.200,123.122,-55.246,-178.898,6.629,148.893
C08270=1155.205,122.873,-55.226,-178.900,6.627,148.893
C08271=1155.209,122.624,-55.206,-178.903,6.625,148.893
C08272=1155.214,122.375,-55.187,-178.906,6.624,148.894
C08273=1155.219,122.126,-55.168,-178.909,6.622,148.894
C08274=1155.223,121.876,-55.148,-178.912,6.620,148.895
C08275=1155.229,121.627,-55.129,-178.914,6.619,148.895
C08276=1155.233,121.378,-55.109,-178.917,6.617,148.896
C08277=1155.238,121.129,-55.090,-178.920,6.615,148.896
C08278=1155.243,120.879,-55.071,-178.922,6.614,148.896
C08279=1155.247,120.630,-55.051,-178.925,6.613,148.897
C08280=1155.253,120.381,-55.032,-178.928,6.611,148.897
C08281=1155.258,120.131,-55.012,-178.930,6.610,148.898
C08282=1155.262,119.883,-54.993,-178.933,6.608,148.898
C08283=1155.267,119.633,-54.974,-178.936,6.606,148.899
C08284=1155.272,119.384,-54.954,-178.939,6.604,148.899
C08285=1155.276,119.135,-54.935,-178.941,6.603,148.899
C08286=1155.281,118.886,-54.916,-178.944,6.601,148.900
C08287=1155.286,118.637,-54.896,-178.947,6.600,148.900
C08288=1155.291,118.387,-54.877,-178.950,6.598,148.901
C08289=1155.296,118.139,-54.858,-178.953,6.596,148.901
C08290=1155.300,117.889,-54.838,-178.955,6.595,148.902
C08291=1155.306,117.640,-54.820,-178.958,6.594,148.902
C08292=1155.310,117.390,-54.801,-178.960,6.592,148.902
C08293=1155.315,117.142,-54.782,-178.963,6.590,148.903
C08294=1155.320,116.892,-54.762,-178.966,6.589,148.903
C08295=1155.324,116.643,-54.743,-178.969,6.587,148.904
C08296=1155.330,116.394,-54.724,-178.972,6.586,148.904
C08297=1155.334,116.144,-54.704,-178.974,6.584,148.905
C08298=1155.339,115.895,-54.686,-178.977,6.582,148.905
C08299=1155.344,115.645,-54.666,-178.979,6.581,148.906
C08300=1155.349,115.397,-54.647,-178.982,6.580,148.906
C08301=1155.353,115.147,-54.628,-178.985,6.578,148.907
C08302=1155.359,114.899,-54.609,-178.988,6.576,148.907
C08303=1155.363,114.649,-54.590,-178.991,6.575,148.907
C08304=1155.368,114.400,-54.571,-178.993,6.573,148.908
C08305=1155.374,114.151,-54.552,-178.996,6.571,148.908
C08306=1155.378,113.902,-54.533,-178.999,6.570,148.909
C08307=1155.383,113.652,-54.514,-179.001,6.569,148.909
C08308=1155.387,113.403,-54.495,-179.004,6.567,148.910
C08309=1155.393,113.154,-54.476,-179.007,6.566,148.910
C08310=1155.397,112.904,-54.457,-179.010,6.564,148.910
C08311=1155.402,112.655,-54.438,-179.012,6.562,148.911
C08312=1155.406,112.406,-54.419,-179.015,6.561,148.911
C08313=1155.412,112.157,-54.400,-179.018,6.559,148.912
C08314=1155.417,111.908,-54.382,-179.020,6.558,148.912
C08315=1155.421,111.658,-54.362,-179.023,6.557,148.913
C08316=1155.427,111.409,-54.343,-179.026,6.555,148.913
C08317=1155.431,111.160,-54.324,-179.028,6.553,148.913
C08318=1155.436,110.911,-54.306,-179.032,6.552,148.914
C08319=1155.441,110.661,-54.287,-179.034,6.550,148.915
C08320=1155.445,110.412,-54.268,-179.037,6.549,148.915
C08321=1155.451,110.163,-54.249,-179.039,6.548,148.915
C08322=1155.455,109.914,-54.230,-179.042,6.546,148.916
C08323=1155.461,109.664,-54.212,-179.045,6.545,148.916
C08324=1155.465,109.415,-54.193,-179.048,6.543,148.917
C08325=1155.470,109.165,-54.174,-179.051,6.541,148.917
C08326=1155.475,108.917,-54.156,-179.053,6.539,148.918
C08327=1155.480,108.667,-54.136,-179.055,6.539,148.918
C08328=1155.484,108.418,-54.118,-179.058,6.537,148.918
C08329=1155.489,108.170,-54.099,-179.061,6.536,148.919
C08330=1155.494,107.919,-54.080,-179.064,6.534,148.919
C08331=1155.499,107.670,-54.062,-179.067,6.532,148.920
C08332=1155.504,107.422,-54.044,-179.070,6.530,148.920
C08333=1155.509,107.171,-54.025,-179.072,6.530,148.921
C08334=1155.513,106.923,-54.006,-179.075,6.528,148.921
C08335=1155.519,106.673,-53.987,-179.078,6.527,148.922
C08336=1155.523,106.424,-53.968,-179.080,6.525,148.922
C08337=1155.528,106.156,-53.949,-179.084,6.523,148.923
C08338=1155.534,105.887,-53.929,-179.086,6.522,148.923
C08339=1155.538,105.619,-53.908,-179.089,6.520,148.924
C08340=1155.544,105.350,-53.888,-179.092,6.519,148.924
C08341=1155.549,105.101,-53.870,-179.095,6.517,148.925
C08342=1155.554,104.852,-53.851,-179.098,6.515,148.925
C08343=1155.558,104.602,-53.833,-179.100,6.514,148.925
C08344=1155.563,104.353,-53.815,-179.103,6.513,148.926
C08345=1155.568,104.104,-53.797,-179.106,6.511,148.927
C08346=1155.574,103.855,-53.778,-179.108,6.510,148.927
C08347=1155.578,103.605,-53.759,-179.111,6.508,148.927
C08348=1155.583,103.356,-53.741,-179.113,6.507,148.928
C08349=1155.588,103.107,-53.722,-179.117,6.506,148.928
C08350=1155.592,102.857,-53.704,-179.119,6.504,148.929
C08351=1155.597,102.608,-53.686,-179.122,6.502,148.929
C08352=1155.602,102.359,-53.668,-179.125,6.501,148.930
C08353=1155.607,102.111,-53.649,-179.127,6.500,148.930
C08354=1155.612,101.860,-53.630,-179.130,6.499,148.931
C08355=1155.617,101.611,-53.612,-179.133,6.497,148.931
C08356=1155.622,101.362,-53.594,-179.135,6.495,148.932
C08357=1155.627,101.113,-53.576,-179.138,6.494,148.932
C08358=1155.632,100.864,-53.557,-179.141,6.493,148.933
C08359=1155.636,100.614,-53.538,-179.144,6.491,148.933
C08360=1155.641,100.365,-53.520,-179.146,6.490,148.933
C08361=1155.646,100.116,-53.502,-179.149,6.488,148.934
C08362=1155.651,99.867,-53.484,-179.152,6.487,148.934
C08363=1155.655,99.617,-53.466,-179.154,6.486,148.935
C08364=1155.661,99.368,-53.447,-179.157,6.484,148.935
C08365=1155.666,99.119,-53.429,-179.160,6.482,148.936
C08366=1155.671,98.869,-53.411,-179.162,6.482,148.936
C08367=1155.675,98.620,-53.393,-179.165,6.480,148.937
C08368=1155.680,98.371,-53.375,-179.168,6.478,148.937
C08369=1155.685,98.121,-53.357,-179.171,6.477,148.938
C08370=1155.690,97.872,-53.339,-179.173,6.476,148.938
C08371=1155.694,97.623,-53.321,-179.176,6.474,148.939
C08372=1155.699,97.374,-53.303,-179.179,6.473,148.939
C08373=1155.705,97.124,-53.284,-179.181,6.471,148.939
C08374=1155.710,96.875,-53.266,-179.184,6.470,148.940
C08375=1155.714,96.625,-53.248,-179.187,6.469,148.941
C08376=1155.719,96.376,-53.230,-179.189,6.467,148.941
C08377=1155.724,96.127,-53.212,-179.192,6.465,148.941
C08378=1155.729,95.878,-53.194,-179.195,6.465,148.942
C08379=1155.734,95.628,-53.176,-179.198,6.463,148.942
C08380=1155.739,95.379,-53.158,-179.200,6.462,148.943
C08381=1155.744,95.130,-53.140,-179.204,6.460,148.944
C08382=1155.749,94.881,-53.122,-179.206,6.459,148.944
C08383=1155.753,94.631,-53.104,-179.208,6.458,148.944
C08384=1155.758,94.382,-53.086,-179.211,6.456,148.945
C08385=1155.763,94.133,-53.068,-179.214,6.455,148.945
C08386=1155.768,93.883,-53.050,-179.216,6.454,148.946
C08387=1155.773,93.634,-53.032,-179.219,6.452,148.946
C08388=1155.778,93.385,-53.014,-179.222,6.450,148.947
C08389=1155.783,93.135,-52.996,-179.225,6.450,148.947
C08390=1155.788,92.886,-52.978,-179.227,6.448,148.948
C08391=1155.793,92.637,-52.960,-179.230,6.446,148.948
C08392=1155.797,92.388,-52.942,-179.233,6.445,148.949
C08393=1155.803,92.138,-52.925,-179.235,6.444,148.949
C08394=1155.808,91.889,-52.907,-179.238,6.443,148.950
C08395=1155.812,91.639,-52.889,-179.241,6.441,148.950
C08396=1155.817,91.390,-52.871,-179.243,6.440,148.951
C08397=1155.821,91.141,-52.853,-179.246,6.439,148.951
C08398=1155.826,90.891,-52.836,-179.249,6.437,148.952
C08399=1155.831,90.642,-52.818,-179.252,6.436,148.952
C08400=1155.836,90.393,-52.800,-179.254,6.435,148.953
C08401=1155.841,90.144,-52.782,-179.257,6.433,148.953
C08402=1155.846,89.894,-52.765,-179.260,6.431,148.953
C08403=1155.851,89.645,-52.747,-179.262,6.431,148.954
C08404=1155.856,89.396,-52.729,-179.265,6.429,148.955
C08405=1155.861,89.146,-52.712,-179.268,6.427,148.955
C08406=1155.865,88.897,-52.694,-179.270,6.427,148.956
C08407=1155.870,88.648,-52.676,-179.273,6.425,148.956
C08408=1155.876,88.398,-52.659,-179.276,6.424,148.956
C08409=1155.880,88.149,-52.641,-179.278,6.423,148.957
C08410=1155.885,87.900,-52.623,-179.281,6.421,148.957
C08411=1155.891,87.650,-52.606,-179.284,6.420,148.958
C08412=1155.895,87.401,-52.589,-179.286,6.419,148.958
C08413=1155.900,87.152,-52.571,-179.289,6.418,148.959
C08414=1155.905,86.902,-52.553,-179.292,6.416,148.959
C08415=1155.910,86.653,-52.535,-179.294,6.415,148.960
C08416=1155.915,86.403,-52.518,-179.297,6.414,148.960
C08417=1155.919,86.154,-52.501,-179.300,6.412,148.961
C08418=1155.925,85.906,-52.483,-179.303,6.410,148.961
C08419=1155.930,85.656,-52.466,-179.306,6.410,148.962
C08420=1155.935,85.407,-52.448,-179.308,6.408,148.962
C08421=1155.939,85.157,-52.431,-179.311,6.406,148.963
C08422=1155.944,84.908,-52.413,-179.313,6.406,148.963
C08423=1155.949,84.658,-52.396,-179.316,6.404,148.964
C08424=1155.954,84.409,-52.378,-179.318,6.403,148.964
C08425=1155.959,84.160,-52.361,-179.321,6.402,148.965
C08426=1155.964,83.910,-52.343,-179.324,6.400,148.965
C08427=1155.969,83.661,-52.326,-179.327,6.399,148.966
C08428=1155.973,83.412,-52.309,-179.329,6.398,148.966
C08429=1155.978,83.162,-52.291,-179.333,6.396,148.967
C08430=1155.984,82.912,-52.274,-179.335,6.396,148.967
C08431=1155.988,82.664,-52.257,-179.337,6.394,148.968
C08432=1155.994,82.414,-52.240,-179.341,6.393,148.968
C08433=1155.998,82.165,-52.222,-179.343,6.392,148.969
C08434=1156.003,81.915,-52.205,-179.345,6.390,148.969
C08435=1156.008,81.666,-52.187,-179.349,6.389,148.970
C08436=1156.013,81.417,-52.170,-179.351,6.388,148.970
C08437=1156.018,81.167,-52.153,-179.354,6.386,148.971
C08438=1156.022,80.918,-52.135,-179.357,6.385,148.971
C08439=1156.028,80.669,-52.118,-179.359,6.384,148.972
C08440=1156.033,80.419,-52.102,-179.362,6.382,148.972
C08441=1156.038,80.151,-52.082,-179.365,6.381,148.973
C08442=1156.043,79.882,-52.064,-179.367,6.380,148.973
C08443=1156.048,79.614,-52.046,-179.370,6.379,148.974
C08444=1156.054,79.345,-52.027,-179.373,6.377,148.974
C08445=1156.058,79.096,-52.010,-179.376,6.376,148.975
C08446=1156.064,78.847,-51.993,-179.378,6.375,148.975
C08447=1156.069,78.598,-51.976,-179.381,6.373,148.976
C08448=1156.074,78.348,-51.959,-179.384,6.372,148.977
C08449=1156.079,78.098,-51.942,-179.386,6.371,148.977
C08450=1156.083,77.850,-51.924,-179.389,6.369,148.977
C08451=1156.089,77.600,-51.907,-179.392,6.369,148.978
C08452=1156.093,77.351,-51.891,-179.395,6.367,148.979
C08453=1156.098,77.101,-51.873,-179.397,6.365,148.979
C08454=1156.103,76.852,-51.856,-179.400,6.365,148.980
C08455=1156.108,76.602,-51.839,-179.403,6.363,148.980
C08456=1156.113,76.354,-51.823,-179.405,6.363,148.981
C08457=1156.118,76.104,-51.805,-179.408,6.361,148.981
C08458=1156.123,75.854,-51.789,-179.411,6.359,148.982
C08459=1156.128,75.605,-51.771,-179.413,6.359,148.982
C08460=1156.133,75.356,-51.755,-179.416,6.357,148.983
C08461=1156.138,75.107,-51.737,-179.418,6.356,148.983
C08462=1156.142,74.857,-51.720,-179.422,6.355,148.984
C08463=1156.148,74.607,-51.703,-179.424,6.353,148.984
C08464=1156.153,74.359,-51.687,-179.426,6.353,148.985
C08465=1156.158,74.109,-51.670,-179.430,6.351,148.985
C08466=1156.162,73.859,-51.653,-179.432,6.350,148.986
C08467=1156.167,73.610,-51.636,-179.435,6.349,148.986
C08468=1156.173,73.361,-51.619,-179.438,6.347,148.987
C08469=1156.177,73.111,-51.603,-179.440,6.346,148.987
C08470=1156.182,72.861,-51.585,-179.443,6.345,148.988
C08471=1156.187,72.613,-51.569,-179.445,6.344,148.988
C08472=1156.192,72.363,-51.552,-179.448,6.343,148.989
C08473=1156.197,72.113,-51.535,-179.451,6.342,148.989
C08474=1156.202,71.864,-51.518,-179.453,6.340,148.990
C08475=1156.207,71.615,-51.502,-179.456,6.339,148.990
C08476=1156.212,71.365,-51.485,-179.459,6.338,148.991
C08477=1156.216,71.116,-51.468,-179.461,6.337,148.991
C08478=1156.222,70.867,-51.451,-179.464,6.336,148.992
C08479=1156.227,70.617,-51.435,-179.467,6.334,148.992
C08480=1156.231,70.368,-51.418,-179.469,6.334,148.993
C08481=1156.237,70.119,-51.401,-179.472,6.332,148.993
C08482=1156.241,69.869,-51.384,-179.475,6.331,148.994
C08483=1156.246,69.620,-51.368,-179.477,6.330,148.994
C08484=1156.252,69.371,-51.351,-179.480,6.328,148.995
C08485=1156.256,69.121,-51.334,-179.482,6.328,148.995
C08486=1156.261,68.872,-51.318,-179.485,6.326,148.996
C08487=1156.266,68.622,-51.302,-179.488,6.325,148.997
C08488=1156.271,68.372,-51.285,-179.491,6.324,148.997
C08489=1156.276,68.124,-51.268,-179.493,6.323,148.998
C08490=1156.281,67.874,-51.252,-179.496,6.322,148.998
C08491=1156.286,67.624,-51.234,-179.498,6.321,148.998
C08492=1156.291,67.376,-51.218,-179.501,6.319,148.999
C08493=1156.296,67.126,-51.202,-179.504,6.318,149.000
C08494=1156.301,66.877,-51.186,-179.507,6.317,149.000
C08495=1156.306,66.627,-51.169,-179.509,6.316,149.001
C08496=1156.311,66.377,-51.152,-179.512,6.315,149.001
C08497=1156.316,66.129,-51.136,-179.515,6.313,149.002
C08498=1156.321,65.879,-51.120,-179.517,6.313,149.002
C08499=1156.326,65.630,-51.103,-179.520,6.311,149.003
C08500=1156.331,65.380,-51.086,-179.522,6.310,149.003
C08501=1156.335,65.131,-51.069,-179.525,6.309,149.004
C08502=1156.341,64.881,-51.054,-179.528,6.308,149.004
C08503=1156.345,64.632,-51.037,-179.530,6.307,149.005
C08504=1156.350,64.383,-51.021,-179.533,6.306,149.005
C08505=1156.355,64.133,-51.004,-179.536,6.304,149.006
C08506=1156.361,63.884,-50.988,-179.538,6.303,149.006
C08507=1156.365,63.634,-50.971,-179.541,6.302,149.007
C08508=1156.370,63.385,-50.955,-179.543,6.301,149.007
C08509=1156.375,63.135,-50.939,-179.546,6.300,149.008
C08510=1156.380,62.886,-50.922,-179.549,6.299,149.009
C08511=1156.385,62.636,-50.907,-179.551,6.297,149.009
C08512=1156.390,62.387,-50.890,-179.554,6.297,149.010
C08513=1156.395,62.138,-50.873,-179.557,6.295,149.010
C08514=1156.400,61.888,-50.857,-179.559,6.294,149.011
C08515=1156.405,61.639,-50.841,-179.562,6.293,149.011
C08516=1156.410,61.389,-50.824,-179.564,6.292,149.012
C08517=1156.415,61.140,-50.809,-179.568,6.291,149.012
C08518=1156.420,60.891,-50.792,-179.570,6.290,149.013
C08519=1156.425,60.641,-50.776,-179.573,6.289,149.013
C08520=1156.430,60.392,-50.760,-179.575,6.288,149.014
C08521=1156.435,60.142,-50.744,-179.578,6.286,149.014
C08522=1156.439,59.893,-50.728,-179.581,6.286,149.015
C08523=1156.445,59.643,-50.712,-179.583,6.284,149.015
C08524=1156.449,59.394,-50.695,-179.586,6.284,149.016
C08525=1156.455,59.144,-50.680,-179.589,6.282,149.016
C08526=1156.459,58.895,-50.663,-179.591,6.281,149.017
C08527=1156.465,58.646,-50.647,-179.594,6.280,149.018
C08528=1156.470,58.397,-50.631,-179.596,6.279,149.018
C08529=1156.474,58.147,-50.615,-179.599,6.278,149.019
C08530=1156.479,57.898,-50.599,-179.602,6.277,149.019
C08531=1156.484,57.648,-50.583,-179.604,6.275,149.020
C08532=1156.489,57.399,-50.567,-179.607,6.275,149.020
C08533=1156.494,57.149,-50.551,-179.610,6.273,149.021
C08534=1156.499,56.900,-50.535,-179.612,6.273,149.021
C08535=1156.505,56.651,-50.519,-179.615,6.271,149.022
C08536=1156.509,56.401,-50.503,-179.618,6.270,149.022
C08537=1156.514,56.152,-50.487,-179.620,6.269,149.023
C08538=1156.519,55.902,-50.471,-179.623,6.268,149.023
C08539=1156.525,55.652,-50.455,-179.625,6.267,149.024
C08540=1156.530,55.404,-50.439,-179.628,6.266,149.024
C08541=1156.534,55.153,-50.423,-179.631,6.265,149.025
C08542=1156.540,54.904,-50.407,-179.633,6.264,149.025
C08543=1156.544,54.655,-50.390,-179.636,6.263,149.026
C08544=1156.550,54.405,-50.375,-179.639,6.261,149.027
C08545=1156.555,54.137,-50.358,-179.641,6.261,149.027
C08546=1156.561,53.868,-50.341,-179.644,6.259,149.028
C08547=1156.566,53.599,-50.323,-179.647,6.258,149.028
C08548=1156.571,53.331,-50.306,-179.650,6.257,149.029
C08549=1156.576,53.081,-50.291,-179.653,6.256,149.029
C08550=1156.580,52.832,-50.275,-179.655,6.255,149.030
C08551=1156.586,52.583,-50.259,-179.658,6.254,149.031
C08552=1156.591,52.333,-50.244,-179.660,6.253,149.031
C08553=1156.596,52.083,-50.228,-179.664,6.252,149.032
C08554=1156.601,51.834,-50.211,-179.666,6.251,149.032
C08555=1156.607,51.585,-50.196,-179.668,6.250,149.033
C08556=1156.611,51.335,-50.180,-179.671,6.249,149.033
C08557=1156.616,51.086,-50.165,-179.673,6.248,149.034
C08558=1156.621,50.836,-50.149,-179.676,6.246,149.034
C08559=1156.626,50.587,-50.133,-179.679,6.246,149.035
C08560=1156.631,50.337,-50.117,-179.682,6.244,149.035
C08561=1156.636,50.088,-50.102,-179.684,6.243,149.036
C08562=1156.641,49.838,-50.086,-179.687,6.243,149.037
C08563=1156.646,49.589,-50.070,-179.689,6.241,149.037
C08564=1156.651,49.339,-50.055,-179.692,6.240,149.037
C08565=1156.656,49.091,-50.039,-179.695,6.239,149.038
C08566=1156.661,48.841,-50.023,-179.697,6.238,149.039
C08567=1156.666,48.591,-50.008,-179.700,6.238,149.039
C08568=1156.671,48.342,-49.992,-179.702,6.236,149.040
C08569=1156.675,48.092,-49.977,-179.705,6.236,149.040
C08570=1156.681,47.843,-49.961,-179.708,6.234,149.041
C08571=1156.686,47.593,-49.945,-179.710,6.233,149.041
C08572=1156.692,47.344,-49.930,-179.713,6.232,149.042
C08573=1156.696,47.094,-49.915,-179.715,6.231,149.042
C08574=1156.701,46.845,-49.899,-179.718,6.230,149.043
C08575=1156.706,46.595,-49.883,-179.721,6.229,149.043
C08576=1156.711,46.346,-49.868,-179.723,6.228,149.044
C08577=1156.716,46.096,-49.852,-179.726,6.227,149.045
C08578=1156.721,45.847,-49.837,-179.729,6.226,149.045
C08579=1156.726,45.598,-49.822,-179.731,6.225,149.046
C08580=1156.731,45.348,-49.806,-179.734,6.224,149.046
C08581=1156.736,45.098,-49.790,-179.736,6.223,149.047
C08582=1156.741,44.849,-49.775,-179.739,6.223,149.047
C08583=1156.746,44.600,-49.760,-179.742,6.221,149.048
C08584=1156.751,44.350,-49.744,-179.744,6.220,149.048
C08585=1156.756,44.101,-49.729,-179.747,6.219,149.049
C08586=1156.761,43.851,-49.713,-179.749,6.218,149.049
C08587=1156.766,43.602,-49.698,-179.752,6.218,149.050
C08588=1156.771,43.353,-49.683,-179.755,6.216,149.051
C08589=1156.776,43.103,-49.667,-179.757,6.215,149.051
C08590=1156.781,42.854,-49.653,-179.760,6.214,149.052
C08591=1156.786,42.603,-49.637,-179.763,6.213,149.052
C08592=1156.791,42.354,-49.621,-179.765,6.213,149.053
C08593=1156.796,42.105,-49.606,-179.768,6.211,149.054
C08594=1156.801,41.856,-49.591,-179.770,6.210,149.054
C08595=1156.806,41.606,-49.576,-179.772,6.210,149.054
C08596=1156.811,41.357,-49.560,-179.776,6.208,149.055
C08597=1156.817,41.107,-49.545,-179.778,6.207,149.056
C08598=1156.821,40.857,-49.530,-179.780,6.207,149.056
C08599=1156.827,40.608,-49.514,-179.783,6.205,149.057
C08600=1156.831,40.359,-49.499,-179.786,6.205,149.057
C08601=1156.837,40.109,-49.484,-179.789,6.203,149.058
C08602=1156.842,39.860,-49.469,-179.791,6.203,149.058
C08603=1156.847,39.610,-49.454,-179.793,6.202,149.059
C08604=1156.852,39.361,-49.439,-179.797,6.201,149.060
C08605=1156.856,39.111,-49.423,-179.799,6.200,149.060
C08606=1156.861,38.861,-49.409,-179.801,6.199,149.061
C08607=1156.867,38.612,-49.393,-179.804,6.198,149.061
C08608=1156.871,38.363,-49.378,-179.807,6.197,149.062
C08609=1156.877,38.113,-49.363,-179.809,6.196,149.062
C08610=1156.882,37.864,-49.348,-179.812,6.195,149.063
C08611=1156.887,37.614,-49.333,-179.814,6.194,149.063
C08612=1156.892,37.365,-49.318,-179.816,6.193,149.064
C08613=1156.897,37.115,-49.303,-179.820,6.192,149.064
C08614=1156.902,36.866,-49.288,-179.822,6.191,149.065
C08615=1156.908,36.617,-49.272,-179.825,6.191,149.066
C08616=1156.912,36.366,-49.257,-179.827,6.189,149.066
C08617=1156.917,36.117,-49.242,-179.830,6.189,149.067
C08618=1156.922,35.867,-49.228,-179.832,6.188,149.067
C08619=1156.927,35.618,-49.213,-179.835,6.186,149.068
C08620=1156.932,35.369,-49.197,-179.837,6.186,149.068
C08621=1156.937,35.119,-49.183,-179.840,6.185,149.069
C08622=1156.943,34.870,-49.167,-179.843,6.183,149.069
C08623=1156.948,34.620,-49.153,-179.846,6.183,149.070
C08624=1156.952,34.371,-49.138,-179.848,6.182,149.071
C08625=1156.958,34.121,-49.122,-179.851,6.181,149.071
C08626=1156.963,33.872,-49.108,-179.853,6.180,149.072
C08627=1156.967,33.623,-49.093,-179.856,6.180,149.072
C08628=1156.973,33.373,-49.078,-179.858,6.178,149.073
C08629=1156.978,33.123,-49.063,-179.861,6.177,149.073
C08630=1156.982,32.874,-49.049,-179.863,6.177,149.074
C08631=1156.988,32.624,-49.033,-179.867,6.175,149.075
C08632=1156.993,32.375,-49.019,-179.869,6.174,149.075
C08633=1156.997,32.126,-49.004,-179.871,6.174,149.076
C08634=1157.003,31.876,-48.989,-179.873,6.173,149.076
C08635=1157.008,31.626,-48.974,-179.876,6.172,149.077
C08636=1157.013,31.377,-48.960,-179.879,6.171,149.077
C08637=1157.018,31.127,-48.944,-179.881,6.170,149.078
C08638=1157.023,30.878,-48.930,-179.884,6.169,149.078
C08639=1157.028,30.628,-48.916,-179.886,6.168,149.079
C08640=1157.033,30.379,-48.900,-179.889,6.168,149.080
C08641=1157.038,30.129,-48.886,-179.892,6.166,149.080
C08642=1157.043,29.880,-48.871,-179.894,6.166,149.081
C08643=1157.048,29.630,-48.857,-179.897,6.165,149.081
C08644=1157.053,29.381,-48.841,-179.899,6.164,149.082
C08645=1157.058,29.131,-48.827,-179.902,6.163,149.082
C08646=1157.063,28.881,-48.812,-179.905,6.162,149.083
C08647=1157.068,28.632,-48.797,-179.907,6.161,149.083
C08648=1157.074,28.382,-48.783,-179.910,6.160,149.084
C08649=1157.079,28.114,-48.767,-179.913,6.160,149.085
C08650=1157.084,27.845,-48.752,-179.915,6.159,149.085
C08651=1157.090,27.576,-48.735,-179.918,6.157,149.086
C08652=1157.096,27.307,-48.720,-179.921,6.157,149.087
C08653=1157.100,27.058,-48.705,-179.924,6.155,149.087
C08654=1157.105,26.808,-48.691,-179.926,6.155,149.088
C08655=1157.110,26.558,-48.677,-179.928,6.154,149.088
C08656=1157.116,26.309,-48.661,-179.931,6.154,149.089
C08657=1157.121,26.059,-48.647,-179.934,6.152,149.089
C08658=1157.126,25.809,-48.633,-179.936,6.151,149.090
C08659=1157.131,25.560,-48.618,-179.939,6.151,149.090
C08660=1157.136,25.311,-48.604,-179.942,6.149,149.091
C08661=1157.141,25.062,-48.589,-179.944,6.148,149.092
C08662=1157.147,24.811,-48.574,-179.947,6.148,149.092
C08663=1157.151,24.562,-48.560,-179.949,6.147,149.093
C08664=1157.156,24.312,-48.546,-179.952,6.146,149.093
C08665=1157.161,24.063,-48.531,-179.954,6.145,149.094
C08666=1157.166,23.813,-48.517,-179.957,6.145,149.095
C08667=1157.172,23.564,-48.503,-179.959,6.144,149.095
C08668=1157.177,23.315,-48.488,-179.962,6.143,149.096
C08669=1157.181,23.065,-48.474,-179.964,6.142,149.096
C08670=1157.186,22.816,-48.459,-179.967,6.141,149.097
C08671=1157.192,22.566,-48.444,-179.969,6.140,149.097
C08672=1157.197,22.316,-48.430,-179.973,6.139,149.098
C08673=1157.202,22.066,-48.416,-179.975,6.138,149.098
C08674=1157.207,21.817,-48.402,-179.977,6.138,149.099
C08675=1157.212,21.568,-48.388,-179.979,6.137,149.100
C08676=1157.217,21.318,-48.373,-179.983,6.136,149.100
C08677=1157.222,21.068,-48.359,-179.985,6.135,149.101
C08678=1157.227,20.818,-48.345,-179.988,6.134,149.101
C08679=1157.232,20.570,-48.330,-179.990,6.134,149.102
C08680=1157.237,20.320,-48.316,-179.992,6.133,149.102
C08681=1157.242,20.071,-48.302,-179.995,6.131,149.103
C08682=1157.247,19.821,-48.287,-179.998,6.131,149.104
C08683=1157.252,19.571,-48.273,-180.000,6.130,149.104
C08684=1157.258,19.322,-48.259,179.997,6.130,149.105
C08685=1157.263,19.073,-48.245,179.995,6.128,149.105
C08686=1157.268,18.823,-48.231,179.992,6.128,149.106
C08687=1157.273,18.573,-48.216,179.990,6.127,149.106
C08688=1157.278,18.324,-48.202,179.987,6.126,149.107
C08689=1157.283,18.074,-48.188,179.985,6.126,149.107
C08690=1157.288,17.825,-48.174,179.982,6.124,149.108
C08691=1157.293,17.575,-48.160,179.980,6.123,149.109
C08692=1157.298,17.325,-48.145,179.977,6.123,149.109
C08693=1157.304,17.076,-48.131,179.975,6.122,149.110
C08694=1157.308,16.827,-48.117,179.972,6.121,149.110
C08695=1157.313,16.577,-48.103,179.969,6.120,149.111
C08696=1157.319,16.326,-48.089,179.967,6.120,149.112
C08697=1157.324,16.077,-48.075,179.965,6.119,149.112
C08698=1157.329,15.828,-48.061,179.962,6.118,149.113
C08699=1157.333,15.578,-48.047,179.959,6.117,149.113
C08700=1157.339,15.329,-48.033,179.956,6.116,149.114
C08701=1157.344,15.080,-48.019,179.954,6.115,149.114
C08702=1157.349,14.830,-48.005,179.952,6.115,149.115
C08703=1157.354,14.580,-47.991,179.950,6.114,149.115
C08704=1157.359,14.331,-47.977,179.946,6.113,149.116
C08705=1157.365,14.081,-47.963,179.944,6.112,149.117
C08706=1157.370,13.831,-47.949,179.941,6.112,149.117
C08707=1157.375,13.582,-47.935,179.939,6.111,149.118
C08708=1157.379,13.333,-47.921,179.937,6.110,149.118
C08709=1157.384,13.083,-47.907,179.934,6.109,149.119
C08710=1157.390,12.833,-47.894,179.931,6.108,149.120
C08711=1157.395,12.584,-47.880,179.929,6.107,149.120
C08712=1157.400,12.334,-47.865,179.926,6.107,149.121
C08713=1157.406,12.085,-47.851,179.924,6.106,149.121
C08714=1157.410,11.836,-47.838,179.922,6.106,149.122
C08715=1157.415,11.585,-47.824,179.919,6.104,149.122
C08716=1157.421,11.336,-47.810,179.916,6.104,149.123
C08717=1157.426,11.087,-47.796,179.914,6.103,149.123
C08718=1157.431,10.837,-47.782,179.911,6.102,149.124
C08719=1157.436,10.588,-47.769,179.909,6.101,149.125
C08720=1157.441,10.338,-47.755,179.907,6.101,149.125
C08721=1157.446,10.088,-47.740,179.904,6.099,149.126
C08722=1157.452,9.838,-47.727,179.901,6.099,149.126
C08723=1157.456,9.589,-47.713,179.898,6.098,149.127
C08724=1157.461,9.340,-47.700,179.896,6.098,149.128
C08725=1157.467,9.090,-47.686,179.894,6.097,149.128
C08726=1157.471,8.840,-47.672,179.891,6.096,149.129
C08727=1157.477,8.591,-47.658,179.888,6.095,149.129
C08728=1157.482,8.341,-47.645,179.886,6.094,149.130
C08729=1157.487,8.092,-47.631,179.883,6.094,149.131
C08730=1157.492,7.842,-47.617,179.881,6.093,149.131
C08731=1157.497,7.592,-47.604,179.879,6.092,149.132
C08732=1157.502,7.343,-47.590,179.876,6.092,149.132
C08733=1157.507,7.094,-47.576,179.873,6.090,149.133
C08734=1157.513,6.844,-47.562,179.871,6.090,149.133
C08735=1157.517,6.594,-47.549,179.868,6.089,149.134
C08736=1157.522,6.344,-47.535,179.866,6.088,149.134
C08737=1157.528,6.095,-47.521,179.863,6.088,149.135
C08738=1157.533,5.845,-47.508,179.861,6.087,149.136
C08739=1157.538,5.596,-47.494,179.859,6.087,149.136
C08740=1157.543,5.346,-47.480,179.856,6.085,149.137
C08741=1157.548,5.097,-47.468,179.853,6.085,149.137
C08742=1157.553,4.847,-47.453,179.851,6.084,149.138
C08743=1157.558,4.597,-47.440,179.848,6.083,149.139
C08744=1157.563,4.348,-47.426,179.846,6.082,149.139
C08745=1157.568,4.098,-47.413,179.844,6.082,149.140
C08746=1157.573,3.849,-47.399,179.841,6.081,149.140
C08747=1157.579,3.599,-47.386,179.839,6.081,149.141
C08748=1157.584,3.350,-47.372,179.836,6.079,149.142
C08749=1157.589,3.100,-47.359,179.833,6.079,149.142
C08750=1157.594,2.851,-47.345,179.831,6.078,149.143
C08751=1157.599,2.601,-47.332,179.829,6.077,149.143
C08752=1157.605,2.351,-47.319,179.826,6.077,149.144
C08753=1157.610,2.082,-47.304,179.824,6.076,149.144
C08754=1157.615,1.812,-47.289,179.820,6.075,149.145
C08755=1157.621,1.543,-47.276,179.818,6.074,149.146
C08756=1157.626,1.274,-47.261,179.816,6.074,149.146
C08757=1157.632,1.024,-47.247,179.813,6.073,149.147
C08758=1157.637,0.775,-47.234,179.810,6.073,149.148
C08759=1157.642,0.525,-47.220,179.808,6.071,149.148
C08760=1157.647,0.275,-47.208,179.805,6.071,149.149
C08761=1157.652,0.026,-47.193,179.803,6.070,149.149
C08762=1157.657,-0.224,-47.181,179.800,6.069,149.150
C08763=1157.663,-0.473,-47.167,179.798,6.069,149.150
C08764=1157.667,-0.723,-47.154,179.795,6.068,149.151
C08765=1157.673,-0.972,-47.141,179.793,6.067,149.151
C08766=1157.677,-1.222,-47.127,179.790,6.067,149.152
C08767=1157.683,-1.471,-47.114,179.788,6.066,149.153
C08768=1157.688,-1.721,-47.101,179.785,6.065,149.153
C08769=1157.693,-1.971,-47.088,179.783,6.064,149.154
C08770=1157.698,-2.220,-47.074,179.780,6.063,149.154
C08771=1157.703,-2.470,-47.061,179.778,6.063,149.155
C08772=1157.709,-2.719,-47.048,179.775,6.062,149.156
C08773=1157.714,-2.969,-47.034,179.773,6.061,149.156
C08774=1157.719,-3.218,-47.021,179.770,6.061,149.157
C08775=1157.724,-3.469,-47.008,179.768,6.060,149.157
C08776=1157.729,-3.718,-46.995,179.766,6.060,149.158
C08777=1157.734,-3.968,-46.981,179.763,6.059,149.158
C08778=1157.739,-4.217,-46.968,179.761,6.058,149.159
C08779=1157.745,-4.467,-46.955,179.758,6.057,149.160
C08780=1157.750,-4.717,-46.942,179.755,6.056,149.160
C08781=1157.755,-4.966,-46.929,179.753,6.056,149.161
C08782=1157.760,-5.216,-46.915,179.751,6.055,149.161
C08783=1157.765,-5.465,-46.903,179.748,6.055,149.162
C08784=1157.771,-5.715,-46.889,179.746,6.054,149.163
C08785=1157.775,-5.965,-46.876,179.743,6.053,149.163
C08786=1157.780,-6.214,-46.864,179.741,6.053,149.164
C08787=1157.786,-6.464,-46.851,179.738,6.052,149.164
C08788=1157.791,-6.714,-46.838,179.736,6.051,149.165
C08789=1157.795,-6.962,-46.824,179.733,6.051,149.166
C08790=1157.801,-7.212,-46.811,179.731,6.050,149.166
C08791=1157.806,-7.462,-46.798,179.729,6.050,149.167
C08792=1157.812,-7.712,-46.785,179.726,6.049,149.167
C08793=1157.816,-7.962,-46.772,179.724,6.048,149.168
C08794=1157.821,-8.211,-46.759,179.721,6.047,149.168
C08795=1157.827,-8.461,-46.746,179.718,6.046,149.169
C08796=1157.832,-8.711,-46.733,179.716,6.046,149.169
C08797=1157.837,-8.960,-46.721,179.713,6.045,149.170
C08798=1157.842,-9.209,-46.708,179.711,6.045,149.171
C08799=1157.847,-9.460,-46.695,179.709,6.044,149.171
C08800=1157.852,-9.709,-46.682,179.706,6.043,149.172
C08801=1157.857,-9.958,-46.669,179.704,6.043,149.172
C08802=1157.862,-10.208,-46.655,179.701,6.042,149.173
C08803=1157.868,-10.457,-46.642,179.699,6.041,149.174
C08804=1157.873,-10.707,-46.630,179.696,6.041,149.174
C08805=1157.878,-10.956,-46.617,179.694,6.040,149.175
C08806=1157.883,-11.206,-46.604,179.691,6.040,149.176
C08807=1157.889,-11.456,-46.592,179.689,6.039,149.176
C08808=1157.894,-11.705,-46.579,179.687,6.038,149.177
C08809=1157.899,-11.956,-46.566,179.684,6.038,149.177
C08810=1157.904,-12.205,-46.553,179.682,6.037,149.178
C08811=1157.909,-12.454,-46.540,179.680,6.036,149.178
C08812=1157.914,-12.704,-46.528,179.677,6.036,149.179
C08813=1157.919,-12.954,-46.515,179.675,6.035,149.179
C08814=1157.925,-13.203,-46.502,179.672,6.035,149.180
C08815=1157.930,-13.453,-46.489,179.670,6.034,149.181
C08816=1157.935,-13.702,-46.476,179.667,6.033,149.181
C08817=1157.939,-13.952,-46.463,179.664,6.032,149.182
C08818=1157.945,-14.201,-46.451,179.662,6.031,149.182
C08819=1157.950,-14.451,-46.438,179.659,6.031,149.183
C08820=1157.956,-14.701,-46.426,179.657,6.030,149.184
C08821=1157.960,-14.951,-46.413,179.654,6.030,149.184
C08822=1157.965,-15.200,-46.400,179.652,6.029,149.185
C08823=1157.971,-15.450,-46.388,179.650,6.028,149.185
C08824=1157.976,-15.699,-46.374,179.647,6.028,149.186
C08825=1157.981,-15.949,-46.361,179.645,6.027,149.187
C08826=1157.986,-16.199,-46.349,179.643,6.026,149.187
C08827=1157.992,-16.448,-46.337,179.640,6.026,149.188
C08828=1157.997,-16.698,-46.324,179.638,6.025,149.188
C08829=1158.002,-16.947,-46.312,179.635,6.025,149.189
C08830=1158.006,-17.197,-46.299,179.633,6.024,149.189
C08831=1158.012,-17.447,-46.286,179.630,6.023,149.190
C08832=1158.018,-17.697,-46.274,179.628,6.023,149.191
C08833=1158.023,-17.946,-46.261,179.625,6.022,149.191
C08834=1158.028,-18.195,-46.249,179.623,6.021,149.192
C08835=1158.032,-18.445,-46.236,179.621,6.021,149.192
C08836=1158.038,-18.695,-46.224,179.618,6.020,149.193
C08837=1158.043,-18.945,-46.211,179.616,6.020,149.194
C08838=1158.048,-19.194,-46.198,179.613,6.019,149.194
C08839=1158.053,-19.444,-46.187,179.611,6.018,149.195
C08840=1158.059,-19.693,-46.174,179.608,6.018,149.195
C08841=1158.064,-19.944,-46.160,179.606,6.017,149.196
C08842=1158.069,-20.193,-46.148,179.603,6.017,149.197
C08843=1158.074,-20.443,-46.136,179.601,6.016,149.197
C08844=1158.080,-20.692,-46.123,179.598,6.016,149.198
C08845=1158.085,-20.941,-46.111,179.596,6.015,149.198
C08846=1158.090,-21.191,-46.099,179.594,6.014,149.199
C08847=1158.095,-21.441,-46.086,179.591,6.014,149.199
C08848=1158.100,-21.691,-46.073,179.589,6.013,149.200
C08849=1158.105,-21.941,-46.061,179.587,6.012,149.201
C08850=1158.110,-22.190,-46.049,179.584,6.012,149.201
C08851=1158.116,-22.440,-46.037,179.582,6.011,149.202
C08852=1158.121,-22.689,-46.024,179.579,6.011,149.202
C08853=1158.126,-22.938,-46.012,179.577,6.010,149.203
C08854=1158.131,-23.188,-46.000,179.574,6.009,149.204
C08855=1158.137,-23.438,-45.987,179.573,6.009,149.204
C08856=1158.142,-23.688,-45.975,179.570,6.009,149.205
C08857=1158.147,-23.957,-45.962,179.567,6.008,149.206
C08858=1158.153,-24.228,-45.948,179.565,6.007,149.206
C08859=1158.159,-24.497,-45.935,179.562,6.006,149.207
C08860=1158.164,-24.767,-45.922,179.559,6.006,149.207
C08861=1158.169,-25.017,-45.909,179.557,6.005,149.208
C08862=1158.174,-25.267,-45.897,179.554,6.005,149.209
C08863=1158.180,-25.516,-45.885,179.552,6.004,149.209
C08864=1158.185,-25.766,-45.873,179.550,6.004,149.210
C08865=1158.190,-26.015,-45.860,179.547,6.003,149.210
C08866=1158.196,-26.265,-45.848,179.545,6.002,149.211
C08867=1158.201,-26.515,-45.836,179.543,6.002,149.211
C08868=1158.205,-26.765,-45.824,179.540,6.001,149.212
C08869=1158.210,-27.014,-45.812,179.537,6.001,149.213
C08870=1158.215,-27.264,-45.800,179.535,6.000,149.213
C08871=1158.220,-27.513,-45.787,179.533,6.000,149.214
C08872=1158.226,-27.763,-45.775,179.531,5.999,149.214
C08873=1158.231,-28.013,-45.763,179.528,5.999,149.215
C08874=1158.236,-28.263,-45.751,179.526,5.998,149.216
C08875=1158.242,-28.513,-45.739,179.523,5.998,149.216
C08876=1158.246,-28.762,-45.727,179.521,5.997,149.217
C08877=1158.252,-29.012,-45.715,179.518,5.997,149.217
C08878=1158.257,-29.261,-45.702,179.516,5.996,149.218
C08879=1158.262,-29.511,-45.690,179.514,5.995,149.219
C08880=1158.268,-29.761,-45.679,179.511,5.995,149.219
C08881=1158.273,-30.010,-45.666,179.509,5.994,149.220
C08882=1158.278,-30.260,-45.654,179.507,5.993,149.220
C08883=1158.283,-30.509,-45.642,179.504,5.993,149.221
C08884=1158.288,-30.759,-45.630,179.502,5.992,149.221
C08885=1158.293,-31.009,-45.618,179.499,5.992,149.222
C08886=1158.299,-31.258,-45.606,179.497,5.991,149.223
C08887=1158.304,-31.508,-45.594,179.495,5.991,149.223
C08888=1158.309,-31.758,-45.582,179.493,5.990,149.224
C08889=1158.314,-32.007,-45.570,179.490,5.990,149.224
C08890=1158.319,-32.257,-45.558,179.488,5.989,149.225
C08891=1158.325,-32.507,-45.546,179.485,5.989,149.226
C08892=1158.330,-32.757,-45.534,179.483,5.988,149.226
C08893=1158.335,-33.006,-45.522,179.480,5.988,149.227
C08894=1158.340,-33.256,-45.510,179.478,5.987,149.227
C08895=1158.345,-33.506,-45.498,179.475,5.986,149.228
C08896=1158.350,-33.755,-45.486,179.473,5.986,149.228
C08897=1158.355,-34.005,-45.475,179.471,5.985,149.229
C08898=1158.361,-34.254,-45.463,179.468,5.984,149.230
C08899=1158.367,-34.504,-45.451,179.466,5.984,149.230
C08900=1158.372,-34.753,-45.439,179.464,5.984,149.231
C08901=1158.376,-35.003,-45.427,179.462,5.984,149.231
C08902=1158.382,-35.253,-45.415,179.459,5.983,149.232
C08903=1158.387,-35.503,-45.403,179.457,5.982,149.233
C08904=1158.392,-35.752,-45.392,179.454,5.982,149.233
C08905=1158.397,-36.002,-45.380,179.452,5.981,149.234
C08906=1158.403,-36.252,-45.368,179.449,5.981,149.235
C08907=1158.408,-36.501,-45.356,179.447,5.980,149.235
C08908=1158.413,-36.751,-45.345,179.444,5.979,149.236
C08909=1158.418,-37.001,-45.333,179.442,5.979,149.236
C08910=1158.424,-37.250,-45.321,179.440,5.979,149.237
C08911=1158.429,-37.499,-45.309,179.438,5.978,149.237
C08912=1158.434,-37.749,-45.297,179.435,5.978,149.238
C08913=1158.439,-37.999,-45.285,179.433,5.977,149.239
C08914=1158.444,-38.249,-45.274,179.430,5.977,149.239
C08915=1158.450,-38.499,-45.262,179.428,5.976,149.240
C08916=1158.455,-38.749,-45.250,179.426,5.975,149.240
C08917=1158.460,-38.998,-45.239,179.423,5.975,149.241
C08918=1158.466,-39.247,-45.227,179.421,5.974,149.242
C08919=1158.471,-39.497,-45.216,179.419,5.974,149.242
C08920=1158.476,-39.747,-45.204,179.416,5.974,149.243
C08921=1158.481,-39.996,-45.192,179.414,5.973,149.243
C08922=1158.486,-40.246,-45.180,179.412,5.973,149.244
C08923=1158.491,-40.496,-45.169,179.409,5.972,149.244
C08924=1158.496,-40.746,-45.157,179.407,5.971,149.245
C08925=1158.502,-40.995,-45.146,179.405,5.971,149.246
C08926=1158.507,-41.245,-45.134,179.402,5.970,149.246
C08927=1158.512,-41.494,-45.123,179.400,5.969,149.247
C08928=1158.517,-41.744,-45.111,179.398,5.970,149.247
C08929=1158.523,-41.994,-45.099,179.395,5.969,149.248
C08930=1158.527,-42.244,-45.087,179.393,5.968,149.249
C08931=1158.533,-42.493,-45.076,179.391,5.968,149.249
C08932=1158.538,-42.743,-45.065,179.388,5.967,149.250
C08933=1158.544,-42.993,-45.053,179.386,5.966,149.250
C08934=1158.548,-43.242,-45.042,179.383,5.966,149.251
C08935=1158.554,-43.492,-45.030,179.381,5.966,149.251
C08936=1158.559,-43.741,-45.019,179.379,5.966,149.252
C08937=1158.564,-43.991,-45.007,179.377,5.965,149.253
C08938=1158.569,-44.241,-44.996,179.374,5.964,149.253
C08939=1158.575,-44.491,-44.984,179.372,5.964,149.254
C08940=1158.580,-44.741,-44.973,179.369,5.963,149.255
C08941=1158.586,-44.990,-44.962,179.367,5.962,149.255
C08942=1158.591,-45.240,-44.950,179.365,5.963,149.256
C08943=1158.596,-45.490,-44.938,179.363,5.962,149.256
C08944=1158.600,-45.739,-44.927,179.360,5.962,149.257
C08945=1158.606,-45.989,-44.916,179.358,5.961,149.257
C08946=1158.611,-46.238,-44.904,179.355,5.960,149.258
C08947=1158.617,-46.488,-44.892,179.353,5.960,149.259
C08948=1158.621,-46.738,-44.881,179.350,5.959,149.259
C08949=1158.628,-46.988,-44.870,179.349,5.959,149.260
C08950=1158.632,-47.237,-44.859,179.346,5.959,149.260
C08951=1158.638,-47.487,-44.847,179.344,5.958,149.261
C08952=1158.642,-47.737,-44.836,179.341,5.958,149.262
C08953=1158.648,-47.986,-44.824,179.339,5.957,149.262
C08954=1158.653,-48.236,-44.813,179.336,5.956,149.263
C08955=1158.659,-48.486,-44.802,179.335,5.956,149.263
C08956=1158.664,-48.736,-44.791,179.333,5.956,149.264
C08957=1158.669,-48.985,-44.780,179.330,5.955,149.264
C08958=1158.674,-49.235,-44.768,179.328,5.954,149.265
C08959=1158.679,-49.484,-44.756,179.325,5.954,149.266
C08960=1158.685,-49.734,-44.746,179.323,5.953,149.266
C08961=1158.691,-50.005,-44.733,179.320,5.953,149.267
C08962=1158.695,-50.275,-44.721,179.318,5.952,149.267
C08963=1158.702,-50.545,-44.709,179.315,5.952,149.268
C08964=1158.707,-50.816,-44.697,179.313,5.951,149.269
C08965=1158.712,-51.066,-44.686,179.311,5.952,149.269
C08966=1158.718,-51.315,-44.674,179.308,5.951,149.270
C08967=1158.723,-51.566,-44.664,179.306,5.950,149.271
C08968=1158.728,-51.815,-44.652,179.304,5.950,149.271
C08969=1158.734,-52.064,-44.641,179.301,5.949,149.272
C08970=1158.739,-52.315,-44.630,179.299,5.948,149.272
C08971=1158.744,-52.565,-44.618,179.297,5.949,149.273
C08972=1158.749,-52.814,-44.607,179.294,5.948,149.273
C08973=1158.754,-53.064,-44.597,179.292,5.948,149.274
C08974=1158.760,-53.314,-44.585,179.290,5.947,149.275
C08975=1158.765,-53.563,-44.574,179.287,5.946,149.275
C08976=1158.770,-53.813,-44.563,179.285,5.946,149.276
C08977=1158.776,-54.063,-44.551,179.283,5.946,149.276
C08978=1158.781,-54.312,-44.541,179.280,5.945,149.277
C08979=1158.786,-54.562,-44.530,179.278,5.944,149.277
C08980=1158.791,-54.812,-44.519,179.276,5.944,149.278
C08981=1158.797,-55.061,-44.507,179.274,5.944,149.279
C08982=1158.802,-55.311,-44.497,179.271,5.944,149.279
C08983=1158.806,-55.561,-44.485,179.269,5.943,149.280
C08984=1158.812,-55.810,-44.475,179.266,5.942,149.280
C08985=1158.817,-56.060,-44.463,179.264,5.942,149.281
C08986=1158.823,-56.309,-44.452,179.262,5.942,149.282
C08987=1158.828,-56.559,-44.442,179.260,5.941,149.282
C08988=1158.832,-56.809,-44.430,179.257,5.941,149.283
C08989=1158.839,-57.059,-44.420,179.255,5.940,149.283
C08990=1158.843,-57.308,-44.408,179.253,5.940,149.284
C08991=1158.848,-57.559,-44.398,179.251,5.940,149.284
C08992=1158.854,-57.808,-44.387,179.248,5.939,149.285
C08993=1158.859,-58.058,-44.376,179.246,5.938,149.286
C08994=1158.865,-58.307,-44.365,179.243,5.938,149.286
C08995=1158.870,-58.557,-44.354,179.241,5.937,149.287
C08996=1158.874,-58.807,-44.343,179.240,5.937,149.287
C08997=1158.880,-59.057,-44.333,179.237,5.937,149.288
C08998=1158.885,-59.306,-44.321,179.235,5.936,149.289
C08999=1158.891,-59.556,-44.311,179.232,5.936,149.289
C09000=1158.896,-59.806,-44.299,179.230,5.935,149.290
C09001=1158.901,-60.055,-44.289,179.228,5.935,149.290
C09002=1158.906,-60.305,-44.278,179.226,5.935,149.291
C09003=1158.912,-60.555,-44.267,179.223,5.934,149.292
C09004=1158.917,-60.804,-44.256,179.221,5.933,149.292
C09005=1158.922,-61.055,-44.245,179.219,5.934,149.293
C09006=1158.927,-61.303,-44.234,179.217,5.933,149.293
C09007=1158.932,-61.554,-44.224,179.214,5.933,149.294
C09008=1158.938,-61.803,-44.213,179.212,5.932,149.294
C09009=1158.943,-62.053,-44.202,179.210,5.932,149.295
C09010=1158.949,-62.303,-44.191,179.207,5.931,149.296
C09011=1158.954,-62.552,-44.180,179.205,5.931,149.296
C09012=1158.959,-62.802,-44.170,179.203,5.930,149.297
C09013=1158.964,-63.052,-44.159,179.200,5.929,149.297
C09014=1158.969,-63.301,-44.148,179.198,5.930,149.298
C09015=1158.974,-63.551,-44.138,179.196,5.929,149.298
C09016=1158.979,-63.802,-44.127,179.193,5.929,149.299
C09017=1158.985,-64.050,-44.116,179.191,5.928,149.300
C09018=1158.990,-64.301,-44.106,179.189,5.928,149.300
C09019=1158.996,-64.551,-44.095,179.187,5.927,149.301
C09020=1159.001,-64.800,-44.084,179.184,5.927,149.302
C09021=1159.006,-65.050,-44.073,179.182,5.926,149.302
C09022=1159.011,-65.300,-44.063,179.181,5.926,149.303
C09023=1159.017,-65.549,-44.052,179.178,5.926,149.303
C09024=1159.022,-65.798,-44.042,179.176,5.925,149.304
C09025=1159.027,-66.049,-44.031,179.173,5.925,149.304
C09026=1159.033,-66.298,-44.020,179.171,5.925,149.305
C09027=1159.038,-66.548,-44.010,179.169,5.924,149.306
C09028=1159.043,-66.797,-43.999,179.167,5.924,149.306
C09029=1159.048,-67.048,-43.989,179.164,5.923,149.307
C09030=1159.053,-67.297,-43.978,179.162,5.923,149.307
C09031=1159.058,-67.547,-43.967,179.160,5.922,149.308
C09032=1159.064,-67.796,-43.957,179.157,5.922,149.308
C09033=1159.069,-68.047,-43.947,179.155,5.921,149.309
C09034=1159.074,-68.296,-43.936,179.153,5.922,149.310
C09035=1159.079,-68.546,-43.925,179.151,5.921,149.310
C09036=1159.085,-68.795,-43.915,179.148,5.920,149.311
C09037=1159.091,-69.045,-43.905,179.146,5.920,149.311
C09038=1159.096,-69.295,-43.894,179.144,5.920,149.312
C09039=1159.101,-69.544,-43.883,179.142,5.919,149.312
C09040=1159.106,-69.794,-43.873,179.140,5.918,149.313
C09041=1159.111,-70.044,-43.862,179.138,5.919,149.314
C09042=1159.116,-70.294,-43.852,179.135,5.918,149.314
C09043=1159.122,-70.544,-43.842,179.133,5.918,149.315
C09044=1159.128,-70.793,-43.831,179.131,5.917,149.315
C09045=1159.132,-71.043,-43.820,179.128,5.917,149.316
C09046=1159.138,-71.292,-43.810,179.126,5.917,149.317
C09047=1159.143,-71.543,-43.799,179.124,5.916,149.317
C09048=1159.149,-71.792,-43.789,179.121,5.915,149.318
C09049=1159.154,-72.042,-43.779,179.120,5.915,149.318
C09050=1159.159,-72.292,-43.768,179.117,5.915,149.319
C09051=1159.165,-72.541,-43.758,179.115,5.914,149.319
C09052=1159.170,-72.792,-43.747,179.113,5.915,149.320
C09053=1159.175,-73.041,-43.737,179.111,5.914,149.321
C09054=1159.181,-73.290,-43.726,179.109,5.913,149.321
C09055=1159.185,-73.540,-43.716,179.106,5.913,149.322
C09056=1159.190,-73.790,-43.706,179.104,5.913,149.322
C09057=1159.196,-74.039,-43.696,179.102,5.912,149.323
C09058=1159.201,-74.289,-43.685,179.099,5.911,149.323
C09059=1159.207,-74.539,-43.675,179.097,5.912,149.324
C09060=1159.212,-74.788,-43.665,179.095,5.911,149.325
C09061=1159.217,-75.039,-43.654,179.093,5.910,149.325
C09062=1159.223,-75.288,-43.644,179.090,5.910,149.326
C09063=1159.228,-75.538,-43.634,179.089,5.910,149.326
C09064=1159.233,-75.788,-43.623,179.086,5.910,149.327
C09065=1159.239,-76.059,-43.613,179.084,5.909,149.327
C09066=1159.245,-76.330,-43.601,179.081,5.908,149.328
C09067=1159.250,-76.602,-43.590,179.078,5.908,149.329
C09068=1159.256,-76.873,-43.579,179.077,5.908,149.329
C09069=1159.261,-77.122,-43.569,179.074,5.908,149.330
C09070=1159.267,-77.372,-43.559,179.072,5.907,149.331
C09071=1159.272,-77.621,-43.549,179.070,5.907,149.331
C09072=1159.277,-77.872,-43.538,179.068,5.907,149.332
C09073=1159.283,-78.121,-43.528,179.066,5.906,149.332
C09074=1159.289,-78.371,-43.518,179.063,5.905,149.333
C09075=1159.293,-78.621,-43.508,179.061,5.905,149.333
C09076=1159.298,-78.870,-43.498,179.059,5.905,149.334
C09077=1159.304,-79.120,-43.488,179.056,5.904,149.335
C09078=1159.309,-79.371,-43.478,179.055,5.904,149.335
C09079=1159.315,-79.620,-43.467,179.052,5.904,149.336
C09080=1159.320,-79.869,-43.458,179.050,5.903,149.336
C09081=1159.325,-80.119,-43.447,179.048,5.903,149.337
C09082=1159.330,-80.369,-43.437,179.046,5.903,149.338
C09083=1159.336,-80.619,-43.427,179.043,5.902,149.338
C09084=1159.341,-80.868,-43.417,179.041,5.902,149.339
C09085=1159.346,-81.118,-43.407,179.039,5.902,149.339
C09086=1159.352,-81.368,-43.397,179.037,5.901,149.340
C09087=1159.357,-81.618,-43.387,179.035,5.901,149.340
C09088=1159.362,-81.867,-43.377,179.033,5.900,149.341
C09089=1159.367,-82.117,-43.367,179.030,5.900,149.342
C09090=1159.373,-82.367,-43.356,179.028,5.899,149.342
C09091=1159.378,-82.617,-43.346,179.026,5.900,149.343
C09092=1159.384,-82.866,-43.337,179.024,5.899,149.343
C09093=1159.389,-83.117,-43.327,179.021,5.898,149.344
C09094=1159.394,-83.366,-43.317,179.019,5.898,149.344
C09095=1159.399,-83.615,-43.307,179.017,5.898,149.345
C09096=1159.405,-83.865,-43.297,179.015,5.897,149.346
C09097=1159.410,-84.116,-43.287,179.013,5.897,149.346
C09098=1159.415,-84.365,-43.277,179.011,5.897,149.347
C09099=1159.420,-84.615,-43.267,179.008,5.896,149.347
C09100=1159.426,-84.864,-43.257,179.006,5.896,149.348
C09101=1159.431,-85.114,-43.248,179.004,5.896,149.348
C09102=1159.436,-85.364,-43.237,179.002,5.895,149.349
C09103=1159.442,-85.614,-43.227,179.000,5.895,149.349
C09104=1159.447,-85.863,-43.218,178.997,5.895,149.350
C09105=1159.452,-86.113,-43.208,178.996,5.895,149.351
C09106=1159.457,-86.363,-43.197,178.994,5.894,149.351
C09107=1159.462,-86.613,-43.188,178.991,5.894,149.352
C09108=1159.468,-86.862,-43.178,178.989,5.894,149.352
C09109=1159.474,-87.112,-43.168,178.987,5.893,149.353
C09110=1159.479,-87.362,-43.159,178.984,5.892,149.354
C09111=1159.484,-87.611,-43.148,178.983,5.892,149.354
C09112=1159.489,-87.862,-43.139,178.980,5.892,149.355
C09113=1159.494,-88.111,-43.129,178.978,5.891,149.355
C09114=1159.500,-88.361,-43.119,178.976,5.891,149.356
C09115=1159.505,-88.611,-43.110,178.974,5.891,149.356
C09116=1159.511,-88.860,-43.100,178.971,5.890,149.357
C09117=1159.515,-89.110,-43.090,178.969,5.891,149.358
C09118=1159.521,-89.360,-43.080,178.967,5.890,149.358
C09119=1159.527,-89.610,-43.070,178.965,5.889,149.359
C09120=1159.531,-89.859,-43.060,178.963,5.889,149.359
C09121=1159.537,-90.109,-43.051,178.961,5.889,149.360
C09122=1159.542,-90.358,-43.041,178.959,5.888,149.360
C09123=1159.548,-90.609,-43.032,178.956,5.888,149.361
C09124=1159.552,-90.859,-43.022,178.954,5.888,149.361
C09125=1159.558,-91.108,-43.011,178.952,5.888,149.362
C09126=1159.563,-91.358,-43.003,178.950,5.887,149.363
C09127=1159.569,-91.607,-42.992,178.948,5.886,149.363
C09128=1159.575,-91.858,-42.983,178.946,5.887,149.364
C09129=1159.579,-92.107,-42.973,178.944,5.886,149.364
C09130=1159.585,-92.357,-42.964,178.941,5.885,149.365
C09131=1159.590,-92.607,-42.954,178.939,5.886,149.365
C09132=1159.596,-92.857,-42.944,178.937,5.885,149.366
C09133=1159.600,-93.106,-42.935,178.936,5.885,149.366
C09134=1159.606,-93.356,-42.924,178.933,5.885,149.367
C09135=1159.611,-93.606,-42.916,178.931,5.884,149.368
C09136=1159.617,-93.855,-42.905,178.929,5.884,149.368
C09137=1159.622,-94.105,-42.896,178.926,5.883,149.369
C09138=1159.628,-94.355,-42.886,178.924,5.883,149.369
C09139=1159.633,-94.605,-42.877,178.922,5.883,149.370
C09140=1159.638,-94.854,-42.867,178.920,5.882,149.371
C09141=1159.643,-95.104,-42.858,178.918,5.882,149.371
C09142=1159.648,-95.354,-42.848,178.916,5.882,149.372
C09143=1159.654,-95.604,-42.839,178.913,5.881,149.372
C09144=1159.660,-95.854,-42.829,178.912,5.881,149.373
C09145=1159.664,-96.103,-42.820,178.909,5.881,149.373
C09146=1159.670,-96.353,-42.811,178.907,5.880,149.374
C09147=1159.675,-96.603,-42.801,178.905,5.880,149.374
C09148=1159.680,-96.853,-42.792,178.903,5.880,149.375
C09149=1159.686,-97.102,-42.781,178.901,5.880,149.376
C09150=1159.691,-97.352,-42.773,178.899,5.879,149.376
C09151=1159.697,-97.602,-42.763,178.896,5.879,149.377
C09152=1159.702,-97.851,-42.753,178.895,5.879,149.377
C09153=1159.708,-98.102,-42.744,178.892,5.878,149.378
C09154=1159.713,-98.351,-42.734,178.890,5.878,149.378
C09155=1159.718,-98.601,-42.725,178.888,5.878,149.379
C09156=1159.724,-98.851,-42.716,178.886,5.877,149.379
C09157=1159.729,-99.100,-42.706,178.884,5.877,149.380
C09158=1159.734,-99.350,-42.697,178.882,5.876,149.381
